// TwinCAT 3 PLC project PLC1
// Company: Nibe Airsite
// ProgramVersion: 3.1.4024.12
// libraries:
//   Tc2_DataExchange, * (Beckhoff Automation GmbH)
//   Tc2_ModbusRTU, * (Beckhoff Automation GmbH)
//   Tc2_ModbusSrv, * (Beckhoff Automation GmbH)
//   Tc2_Standard, * (Beckhoff Automation GmbH)
//   Tc2_SUPS, * (Beckhoff Automation GmbH)
//   Tc2_System, * (Beckhoff Automation GmbH)
//   Tc2_SystemCX, * (Beckhoff Automation GmbH)
//   Tc2_TcpIp, * (Beckhoff Automation GmbH)
//   Tc2_Utilities, * (Beckhoff Automation GmbH)
//   Tc3_BA_Common, * (Beckhoff Automation GmbH)
//   Tc3_JsonXml, * (Beckhoff Automation GmbH)
//   Tc3_Module, * (Beckhoff Automation GmbH)
// project tree:
//   DUTs/Alarms/ AlarmDef.TcDUT, AlarmHandler.TcPOU, AlarmPolarity.TcDUT, AlarmPriority.TcDUT, AlarmLog.TcDUT, AlarmMonitor.TcPOU, AlarmEvent.TcDUT
//   DUTs/Custom/ExtraAlarms/ AdsTagsExtraAlarms.TcDUT, GreenMasterStatusExtraAlarms.TcDUT, ExtraAlarms_Interface.TcPOU
//   DUTs/Custom/ParallelUnits/ AdsTagsParallelUnits.TcDUT, ParallelUnits.TcPOU, ParallelUnitsSettings.TcDUT, ParallelUnitsStatus.TcDUT, RemoteOrder.TcDUT, RemoteStatusData.TcDUT
//   DUTs/Custom/SmokeControl/ AdsTagsSmokeControl.TcDUT, SmokeControl_Interface.TcPOU, GreenMasterStatusSmokeControl.TcDUT, SxDuoInterface.TcDUT
//   DUTs/Custom/Redundancy/ TagsRedundancy.TcDUT (not stored), adsValue_AggStat.TcPOU, AggStat.TcDUT, RedundancyStatus.TcDUT, RedundancySettings.TcDUT (not stored), Redundancy.TcPOU
//   DUTs/Custom/_Standard/ AdsTags.TcDUT, GreenMasterSettings.TcDUT, GreenMasterStatus.TcDUT, Standard_Interface.TcPOU, TimeChannel_CT_CF.TcDUT
//   DUTs/Defrost/ DefrostSections.TcDUT, Defrost.TcPOU, DefrostStates.TcDUT
//   DUTs/Exercise/ ExerciseF_QM2.TcPOU, ExerciseF_P1.TcPOU
//   DUTs/GreenMaster/ SystemStatesRunMode.TcDUT, SystemStatesRunModeExternal.TcDUT, GreenMasterXXL.TcPOU, GreenMasterBase.TcPOU, SystemStates.TcDUT
//   DUTs/IO/ AI3468.TcDUT, AnalogInput.TcPOU, FlowInput.TcPOU, TemperatureInput.TcPOU, AnalogOutput.TcPOU, AnalogSwitch.TcPOU, DigitalInput.TcPOU, DigitalOutput.TcPOU, BaseIO.TcPOU, PressureInput.TcPOU, TIoKind.TcDUT
//   DUTs/ModbusRTU/ EBM_Speed.TcPOU, Gebhardt_Power.TcPOU, Gebhardt_Speed.TcPOU, ModbusReadWordArray.TcPOU, EBM_Power.TcPOU, Modbus.TcPOU, ModbusIo.TcPOU, ModbusWriteBits.TcPOU, ModbusWriteWord.TcPOU, ModbusRegisterType.TcDUT, ModbusRTU.TcPOU, ModbusReadWord.TcPOU, ModbusReadBits.TcPOU
//   DUTs/Parameters/Alarm/ AlarmControl.TcDUT, AlarmDelays.TcDUT, AlarmLimits.TcDUT, AlarmLimitsA.TcDUT, AlarmLimitsB.TcDUT, AlarmLimitsC.TcDUT, AlarmParameters.TcDUT, AlarmParametersFB.TcPOU (not stored), AlarmsA.TcDUT, AlarmsB.TcDUT, AlarmsC.TcDUT, AlarmsDelaysA.TcDUT, AlarmsDelaysB.TcDUT, AlarmsDelaysC.TcDUT, AlarmSignals.TcDUT
//   DUTs/Controllers/ Band.TcPOU, BandLimit.TcPOU, Controller.TcPOU, PidController.TcPOU, InterpolateNewton.TcPOU, Interpolate.TcPOU, Ramp.TcPOU
//   DUTs/Controls/ SupplyAirControl.TcPOU, ExtractAirControl.TcPOU
//   DUTs/Dampers/ BaseDamper.TcPOU, Damper.TcPOU, DamperMonitor.TcPOU
//   DUTs/Events/ Event.TcDUT, EventLog.TcPOU, EventLogData.TcDUT, EventTypes.TcDUT
//   DUTs/Fans/ Fan.TcPOU, FanControl.TcPOU, FanControlTypes.TcDUT, PostVentilation.TcPOU, PressureToFlow.TcPOU, SpecificFanPower.TcPOU
//   DUTs/Fire/ FireDamper.TcPOU, SmokeDetector.TcPOU
//   DUTs/GreenMaster/IO/ GreenMasterAIU_Base.TcPOU, GreenMasterAIU_ModbusRTU.TcPOU, GreenMasterAI_Base.TcPOU, GreenMasterAO_Base.TcPOU, GreenMasterDI_Base.TcPOU, GreenMasterDO_Base.TcPOU, GreenMasterSmokeControl.TcPOU, GreenMasterSmokeControl_Base.TcPOU, GreenMasterAI.TcPOU, GreenMasterAIU.TcPOU, GreenMasterAO.TcPOU, GreenMasterDI.TcPOU, GreenMasterDO.TcPOU
//   DUTs/ModbusTCP/ ModbusTCP.TcPOU
//   DUTs/Parameters/ GreenMasterBaseParameters.TcDUT, GreenMasterBaseParametersFB.TcPOU, GreenMasterParametersXXL.TcDUT, GreenMasterParametersXXLFB.TcDUT
//   DUTs/Parameters/IO/ AnalogInputParameters.TcDUT, AnalogInputParametersFB.TcPOU, AnalogOutputCalibration.TcDUT, AnalogOutputCalibrationParameters.TcDUT, AnalogOutputOverrideParameters.TcDUT, AnalogOutputParameters.TcDUT, AnalogOutputParametersFB.TcPOU, DigitalInputParameters.TcDUT, DigitalInputParametersFB.TcPOU, DigitalOutputOverrideParameters.TcDUT, DigitalOutputParameters.TcDUT, DigitalOutputParametersFB.TcPOU, InputStatus.TcDUT, IoParameters.TcDUT, IOParametersFB.TcPOU, IoStatus.TcDUT, SensorStatus.TcDUT, SmokeControlStatus.TcDUT
//   DUTs/Parameters/Redundancy/ RedundancyParameters.TcDUT
//   DUTs/Parameters/Regulation/ AirParameters.TcDUT, AirParametersFB.TcPOU, ColdRecyclingParameters.TcDUT, ControllerParameters.TcDUT, DefaultParameters.TcDUT, DefaultParametersFB.TcPOU, FanTypes.TcDUT, FireParameters.TcDUT, HeaterOutputDirections.TcDUT, RegulationControlParameters.TcDUT, RegulationParameters.TcDUT, RegulationParametersFB.TcPOU, SetPointAdjustment.TcDUT, SetPointAdjustmentFB.TcPOU, SetPointOffsetCurve.TcDUT, TemperatureCompensationSources.TcDUT, TemperatureControlParameters.TcDUT, TemperatureControlParametersFB.TcPOU, TemperatureControlSources.TcDUT
//   DUTs/Parameters/Simulation/ SimulateFlow.TcPOU, SimulationFB.TcPOU, SimulationParameters.TcDUT, SimulationParametersFB.TcPOU
//   DUTs/Parameters/SmokeControl/ NetLinkParameters.TcDUT, NetLinkParametersFB.TcPOU, SmokeControlExerciseParameters.TcDUT, SmokeControlFireParameters.TcDUT, SmokeControlParametersBase.TcDUT, SmokeControlParametersBaseFB.TcPOU, SxDuoCommand.TcDUT, SxDuoParameters.TcDUT, SxDuoParametersFB.TcPOU, SxDuoStatus.TcDUT, SxDuoUnit.TcDUT, SxDuoUnitFB.TcPOU
//   DUTs/Parameters/System/Defrost/ DefrostParameters.TcDUT, DefrostStageParameters.TcDUT, SetPointReductionParameters.TcDUT, WinterShutdownParameters.TcDUT
//   DUTs/Parameters/System/Exercise/ ExerciseCirculationPumpsParameters.TcDUT, ExerciseCirculationPumpsParametersFB.TcPOU, ExerciseExternalFireControlParameters.TcDUT, ExerciseExternalFireControlParametersFB.TcPOU, ExerciseFireBypassDamperParameters.TcDUT, ExerciseFireBypassDamperParametersFB.TcPOU, ExerciseParameters.TcDUT, ExerciseParametersFB.TcPOU
//   DUTs/Parameters/System/Operation/ AlternativeOperation.TcDUT, CoolingRecycling.TcDUT, DIStartUnit.TcDUT, LocalTimeControl.TcDUT, MaxFilterPressure.TcDUT, NightReduction.TcDUT, OperationParametersFB.TcPOU, OvkActivation.TcDUT, RecirculationControl.TcDUT, RelativeHumidity.TcDUT, SetPointTypes.TcDUT, StartControl.TcDUT, StartupFanDelay.TcDUT, StartupRecycling.TcDUT, SystemOperationParameters.TcDUT, SystemOperationParametersXXL.TcDUT, TimeChannelDayParameters.TcDUT, TimeChannelParameters.TcDUT, TimeChannelParametersFB.TcPOU, TimeChannelDayParametersFB.TcPOU, UnitOperation.TcDUT
//   DUTs/Parameters/System/ SystemParameters.TcDUT, SystemParametersFB.TcPOU, SystemParametersXXL.TcDUT
//   DUTs/Smoke Control/ DamperControl.TcPOU, DamperModule.TcPOU
//   DUTs/System/ AnyEqual.TcPOU, Permissions.TcDUT, Supervisor.TcPOU, User.TcDUT
//   DUTs/Utilities/ ActuatorMonitor.TcPOU, AnalogMultiplexer.TcPOU, Average.TcPOU, DeviationMonitor.TcPOU, DeviationMonitorMode.TcDUT, CalculateEfficiency.TcPOU, ifc_int.TcPOU, ifc_bool.TcPOU, ifc_lreal.TcPOU, LREAL_BMUX.TcPOU, BOOL_BMUX.TcPOU, BoolToErrorText.TcPOU, DigitalSignal.TcPOU, EMA.TcPOU, GetBit.TcPOU, GetTickCount.TcPOU, Hysteresis.TcPOU, LimitValue.TcPOU, MAX_FB.TcPOU, MIN_FB.TcPOU, NowDT.TcPOU, PulseCounter.TcPOU, PWM.TcPOU, REAL_TO_WORD_SAFE.TcPOU, LREAL_TO_WORD_SAFE.TcPOU, Scale.TcPOU, SetBit.TcPOU, TimeChannel1CH.TcPOU, TimeChannel1CH_Data.TcDUT, TimeChannelSettings.TcDUT, Timer.TcPOU, TimerDays.TcDUT, WriteBoolIf.TcPOU, WriteLRealIf.TcPOU, WriteLRealOnlyIf.TcPOU
//   DUTs/Valves/ BaseValve.TcPOU, Valve.TcPOU, ValveMonitor.TcPOU
//   DUTs/Ventilation/ FB_GM_NIGHTCOOL.TcPOU, VentilationControl.TcPOU
//   GVLs/ ADS_ParallelUnits.TcGVL, ADS_SmokeControl.TcGVL, ADS_Standard.TcGVL, ADS_ExtraAlarms.TcGVL, AnalogInputs.TcDUT, AnalogOutputs.TcDUT, DigitalInputs.TcDUT, DigitalInputLevels.TcDUT, DigitalOutputs.TcDUT, ComponentNames.TcDUT, ExtraAlarmInputs.TcGVL, GetComponent.TcPOU, Globals.TcGVL, GVL.TcGVL, GVL_Redundancy.TcGVL, IOTypes.TcDUT, GlobalSettings.TcGVL, Component.TcDUT, ModbusRTU_IO.TcDUT
//   / PlcTask.TcTTO, Task_4.TcTTO
//   POUs/ AdsWriteVariable.TcPOU, GreenMasterXXL_FB.TcPOU, Main.TcPOU, SimpleTimeChannel.TcPOU, SmokeControl.TcPOU, AdsReadVariable.TcPOU, TestPID.TcPOU, Timers.TcPOU
// real-time tasks:
//   TASK PlcTask: cycle T#50000us, priority 20, ADS port 350
//   TASK Task 4: cycle T#10ms, priority 1, ADS port 351
// I/O:
//   DEVICE Device 1 (Beckhoff CCAT)
//   DEVICE Device CTH (CX-BK) (disabled)
//     Box CTH (CX-BK)
//   DEVICE Device STD (CX-BK)
//     Box STD (CX-BK)
//   DEVICE Device GMA (CX-BK) (disabled)
//     Box STD (CX-BK)
// variable links:
//   PLC1/PLC1 Instance <-> Device CTH (CX-BK)/Box CTH (CX-BK)
//     PlcTask Inputs/Globals.IO.AIn.AI01_Error <-> AI 2.1 (KL3208-0010-4)/Channel 1/State @bit 6
//     PlcTask Inputs/Globals.IO.AIn.AI02_Error <-> AI 2.1 (KL3208-0010-4)/Channel 2/State @bit 6
//     PlcTask Inputs/Globals.IO.AIn.AI03_Error <-> AI 2.1 (KL3208-0010-4)/Channel 3/State @bit 6
//     PlcTask Inputs/Globals.IO.AIn.AI04_Error <-> AI 2.1 (KL3208-0010-4)/Channel 4/State @bit 6
//     PlcTask Inputs/Globals.IO.AIn.AI05_Error <-> AI 2.2 (KL3208-0010-4)/Channel 1/State @bit 6
//     PlcTask Inputs/Globals.IO.AIn.AI06_Error <-> AI 2.2 (KL3208-0010-4)/Channel 2/State @bit 6
//     PlcTask Inputs/Globals.IO.AIn.AI07_Error <-> AI 2.2 (KL3208-0010-4)/Channel 3/State @bit 6
//     PlcTask Inputs/Globals.IO.AIn.AI08_Error <-> AI 2.2 (KL3208-0010-4)/Channel 4/State @bit 6
//     PlcTask Inputs/Globals.IO.AIn.AI09_Error <-> AI 3.1 (KL3208-0010-4)/Channel 1/State @bit 6
//     PlcTask Inputs/Globals.IO.AIn.AI10_Error <-> AI 3.1 (KL3208-0010-4)/Channel 2/State @bit 6
//     PlcTask Inputs/Globals.IO.AIn.AI11_Error <-> AI 3.1 (KL3208-0010-4)/Channel 3/State @bit 6
//     PlcTask Inputs/Globals.IO.AIn.AI12_Error <-> AI 3.1 (KL3208-0010-4)/Channel 4/State @bit 6
//     PlcTask Inputs/Globals.IO.AIn.AI13_Error <-> AI 3.2 (KL3208-0010-4)/Channel 1/State @bit 6
//     PlcTask Inputs/Globals.IO.AIn.AI14_Error <-> AI 3.2 (KL3208-0010-4)/Channel 2/State @bit 6
//     PlcTask Inputs/Globals.IO.AIn.AI15_Error <-> AI 3.2 (KL3208-0010-4)/Channel 3/State @bit 6
//     PlcTask Inputs/Globals.IO.AIn.AI16_Error <-> AI 3.2 (KL3208-0010-4)/Channel 4/State @bit 6
//     PlcTask Inputs/Globals.IO.AIn.AI17_Error <-> AI 4.1 (KL3468-4)/Channel 1/State @bit 6
//     PlcTask Inputs/Globals.IO.AIn.AI18_Error <-> AI 4.1 (KL3468-4)/Channel 2/State @bit 6
//     PlcTask Inputs/Globals.IO.AIn.AI19_Error <-> AI 4.1 (KL3468-4)/Channel 3/State @bit 6
//     PlcTask Inputs/Globals.IO.AIn.AI20_Error <-> AI 4.1 (KL3468-4)/Channel 4/State @bit 6
//     PlcTask Inputs/Globals.IO.AIn.AI21_Error <-> AI 4.2 (KL3468-4)/Channel 1/State @bit 6
//     PlcTask Inputs/Globals.IO.AIn.AI22_Error <-> AI 4.2 (KL3468-4)/Channel 2/State @bit 6
//     PlcTask Inputs/Globals.IO.AIn.AI23_Error <-> AI 4.2 (KL3468-4)/Channel 3/State @bit 6
//     PlcTask Inputs/Globals.IO.AIn.AI24_Error <-> AI 4.2 (KL3468-4)/Channel 4/State @bit 6
//     PlcTask Inputs/Globals.IO.DIn.DI01 <-> DI 1 (KL1408)/Channel 1/Input
//     PlcTask Inputs/Globals.IO.DIn.DI02 <-> DI 1 (KL1408)/Channel 2/Input
//     PlcTask Inputs/Globals.IO.DIn.DI03 <-> DI 1 (KL1408)/Channel 3/Input
//     PlcTask Inputs/Globals.IO.DIn.DI04 <-> DI 1 (KL1408)/Channel 4/Input
//     PlcTask Inputs/Globals.IO.DIn.DI05 <-> DI 1 (KL1408)/Channel 5/Input
//     PlcTask Inputs/Globals.IO.DIn.DI06 <-> DI 1 (KL1408)/Channel 6/Input
//     PlcTask Inputs/Globals.IO.DIn.DI07 <-> DI 1 (KL1408)/Channel 7/Input
//     PlcTask Inputs/Globals.IO.DIn.DI08 <-> DI 1 (KL1408)/Channel 8/Input
//     PlcTask Inputs/Globals.IO.DIn.DI09 <-> DI 2 (KL1408)/Channel 1/Input
//     PlcTask Inputs/Globals.IO.DIn.DI10 <-> DI 2 (KL1408)/Channel 2/Input
//     PlcTask Inputs/Globals.IO.DIn.DI11 <-> DI 2 (KL1408)/Channel 3/Input
//     PlcTask Inputs/Globals.IO.DIn.DI12 <-> DI 2 (KL1408)/Channel 4/Input
//     PlcTask Inputs/Globals.IO.DIn.DI13 <-> DI 2 (KL1408)/Channel 5/Input
//     PlcTask Inputs/Globals.IO.DIn.DI14 <-> DI 2 (KL1408)/Channel 6/Input
//     PlcTask Inputs/Globals.IO.DIn.DI15 <-> DI 2 (KL1408)/Channel 7/Input
//     PlcTask Inputs/Globals.IO.DIn.DI16 <-> DI 2 (KL1408)/Channel 8/Input
//     PlcTask Inputs/Globals.IO.DIn.DI17 <-> DI 3 (KL1408)/Channel 1/Input
//     PlcTask Inputs/Globals.IO.DIn.DI18 <-> DI 3 (KL1408)/Channel 2/Input
//     PlcTask Inputs/Globals.IO.DIn.DI19 <-> DI 3 (KL1408)/Channel 3/Input
//     PlcTask Inputs/Globals.IO.DIn.DI20 <-> DI 3 (KL1408)/Channel 4/Input
//     PlcTask Inputs/Globals.IO.DIn.DI21 <-> DI 3 (KL1408)/Channel 5/Input
//     PlcTask Inputs/Globals.IO.DIn.DI22 <-> DI 3 (KL1408)/Channel 6/Input
//     PlcTask Inputs/Globals.IO.DIn.DI23 <-> DI 3 (KL1408)/Channel 7/Input
//     PlcTask Inputs/Globals.IO.DIn.DI24 <-> DI 3 (KL1408)/Channel 8/Input
//     PlcTask Outputs/Globals.IO.AOut.AO01 <-> AO 1.1 (KL4408-4)/Channel 1/Data Out
//     PlcTask Outputs/Globals.IO.AOut.AO02 <-> AO 1.1 (KL4408-4)/Channel 2/Data Out
//     PlcTask Outputs/Globals.IO.AOut.AO03 <-> AO 1.1 (KL4408-4)/Channel 3/Data Out
//     PlcTask Outputs/Globals.IO.AOut.AO04 <-> AO 1.1 (KL4408-4)/Channel 4/Data Out
//     PlcTask Outputs/Globals.IO.AOut.AO05 <-> AO 1.2 (KL4408-4)/Channel 1/Data Out
//     PlcTask Outputs/Globals.IO.AOut.AO06 <-> AO 1.2 (KL4408-4)/Channel 2/Data Out
//     PlcTask Outputs/Globals.IO.AOut.AO07 <-> AO 1.2 (KL4408-4)/Channel 3/Data Out
//     PlcTask Outputs/Globals.IO.AOut.AO08 <-> AO 1.2 (KL4408-4)/Channel 4/Data Out
//     PlcTask Outputs/Globals.IO.DOut.DO01 <-> DO 1 (KL2408)/Channel 1/Output
//     PlcTask Outputs/Globals.IO.DOut.DO02 <-> DO 1 (KL2408)/Channel 2/Output
//     PlcTask Outputs/Globals.IO.DOut.DO03 <-> DO 1 (KL2408)/Channel 3/Output
//     PlcTask Outputs/Globals.IO.DOut.DO04 <-> DO 1 (KL2408)/Channel 4/Output
//     PlcTask Outputs/Globals.IO.DOut.DO05 <-> DO 1 (KL2408)/Channel 5/Output
//     PlcTask Outputs/Globals.IO.DOut.DO06 <-> DO 1 (KL2408)/Channel 6/Output
//     PlcTask Outputs/Globals.IO.DOut.DO07 <-> DO 1 (KL2408)/Channel 7/Output
//     PlcTask Outputs/Globals.IO.DOut.DO08 <-> DO 1 (KL2408)/Channel 8/Output
//     PlcTask Outputs/Globals.IO.DOut.DO09 <-> DO 2 (KL2408)/Channel 1/Output
//     PlcTask Outputs/Globals.IO.DOut.DO10 <-> DO 2 (KL2408)/Channel 2/Output
//     PlcTask Outputs/Globals.IO.DOut.DO11 <-> DO 2 (KL2408)/Channel 3/Output
//     PlcTask Outputs/Globals.IO.DOut.DO12 <-> DO 2 (KL2408)/Channel 4/Output
//     PlcTask Outputs/Globals.IO.DOut.DO13 <-> DO 2 (KL2408)/Channel 5/Output
//     PlcTask Outputs/Globals.IO.DOut.DO14 <-> DO 2 (KL2408)/Channel 6/Output
//     PlcTask Outputs/Globals.IO.DOut.DO15 <-> DO 2 (KL2408)/Channel 7/Output
//     PlcTask Outputs/Globals.IO.DOut.DO16 <-> DO 2 (KL2408)/Channel 8/Output
//     PlcTask Outputs/Globals.IO.DOut.RDO01 <-> RDO 1 (KL2652)/Channel 1/Output
//     PlcTask Outputs/Globals.IO.DOut.RDO02 <-> RDO 1 (KL2652)/Channel 2/Output
//     PlcTask Outputs/Globals.IO.DOut.RDO03 <-> RDO 2 (KL2652)/Channel 1/Output
//     PlcTask Outputs/Globals.IO.DOut.RDO04 <-> RDO 2 (KL2652)/Channel 2/Output
//   PLC1/PLC1 Instance <-> Device GMA (CX-BK)/Box STD (CX-BK)
//     PlcTask Inputs/Globals.IO.AIn.AI01_Error <-> AI 2.1 (KL3208-0010-4)/Channel 1/State @bit 6
//     PlcTask Inputs/Globals.IO.AIn.AI02_Error <-> AI 2.1 (KL3208-0010-4)/Channel 2/State @bit 6
//     PlcTask Inputs/Globals.IO.AIn.AI03_Error <-> AI 2.1 (KL3208-0010-4)/Channel 3/State @bit 6
//     PlcTask Inputs/Globals.IO.AIn.AI04_Error <-> AI 2.1 (KL3208-0010-4)/Channel 4/State @bit 6
//     PlcTask Inputs/Globals.IO.AIn.AI05_Error <-> AI 2.2 (KL3208-0010-4)/Channel 1/State @bit 6
//     PlcTask Inputs/Globals.IO.AIn.AI06_Error <-> AI 2.2 (KL3208-0010-4)/Channel 2/State @bit 6
//     PlcTask Inputs/Globals.IO.AIn.AI07_Error <-> AI 2.2 (KL3208-0010-4)/Channel 3/State @bit 6
//     PlcTask Inputs/Globals.IO.AIn.AI08_Error <-> AI 2.2 (KL3208-0010-4)/Channel 4/State @bit 6
//     PlcTask Inputs/Globals.IO.DIn.DI01 <-> DI 1 (KL1408)/Channel 1/Input
//     PlcTask Inputs/Globals.IO.DIn.DI02 <-> DI 1 (KL1408)/Channel 2/Input
//     PlcTask Inputs/Globals.IO.DIn.DI03 <-> DI 1 (KL1408)/Channel 3/Input
//     PlcTask Inputs/Globals.IO.DIn.DI04 <-> DI 1 (KL1408)/Channel 4/Input
//     PlcTask Inputs/Globals.IO.DIn.DI05 <-> DI 1 (KL1408)/Channel 5/Input
//     PlcTask Inputs/Globals.IO.DIn.DI06 <-> DI 1 (KL1408)/Channel 6/Input
//     PlcTask Inputs/Globals.IO.DIn.DI07 <-> DI 1 (KL1408)/Channel 7/Input
//     PlcTask Inputs/Globals.IO.DIn.DI08 <-> DI 1 (KL1408)/Channel 8/Input
//     PlcTask Inputs/Globals.IO.DIn.DI09 <-> DI 2 (KL1408)/Channel 1/Input
//     PlcTask Inputs/Globals.IO.DIn.DI10 <-> DI 2 (KL1408)/Channel 2/Input
//     PlcTask Inputs/Globals.IO.DIn.DI11 <-> DI 2 (KL1408)/Channel 3/Input
//     PlcTask Inputs/Globals.IO.DIn.DI12 <-> DI 2 (KL1408)/Channel 4/Input
//     PlcTask Inputs/Globals.IO.DIn.DI13 <-> DI 2 (KL1408)/Channel 5/Input
//     PlcTask Inputs/Globals.IO.DIn.DI14 <-> DI 2 (KL1408)/Channel 6/Input
//     PlcTask Inputs/Globals.IO.DIn.DI15 <-> DI 2 (KL1408)/Channel 7/Input
//     PlcTask Inputs/Globals.IO.DIn.DI16 <-> DI 2 (KL1408)/Channel 8/Input
//     PlcTask Outputs/Globals.IO.AOut.AO01 <-> AO 1.1 (KL4408-4)/Channel 1/Data Out
//     PlcTask Outputs/Globals.IO.AOut.AO02 <-> AO 1.1 (KL4408-4)/Channel 2/Data Out
//     PlcTask Outputs/Globals.IO.AOut.AO03 <-> AO 1.1 (KL4408-4)/Channel 3/Data Out
//     PlcTask Outputs/Globals.IO.AOut.AO04 <-> AO 1.1 (KL4408-4)/Channel 4/Data Out
//     PlcTask Outputs/Globals.IO.AOut.AO05 <-> AO 1.2 (KL4408-4)/Channel 1/Data Out
//     PlcTask Outputs/Globals.IO.AOut.AO06 <-> AO 1.2 (KL4408-4)/Channel 2/Data Out
//     PlcTask Outputs/Globals.IO.AOut.AO07 <-> AO 1.2 (KL4408-4)/Channel 3/Data Out
//     PlcTask Outputs/Globals.IO.AOut.AO08 <-> AO 1.2 (KL4408-4)/Channel 4/Data Out
//     PlcTask Outputs/Globals.IO.DOut.DO01 <-> DO 1 (KL2408)/Channel 1/Output
//     PlcTask Outputs/Globals.IO.DOut.DO02 <-> DO 1 (KL2408)/Channel 2/Output
//     PlcTask Outputs/Globals.IO.DOut.DO03 <-> DO 1 (KL2408)/Channel 3/Output
//     PlcTask Outputs/Globals.IO.DOut.DO04 <-> DO 1 (KL2408)/Channel 4/Output
//     PlcTask Outputs/Globals.IO.DOut.DO05 <-> DO 1 (KL2408)/Channel 5/Output
//     PlcTask Outputs/Globals.IO.DOut.DO06 <-> DO 1 (KL2408)/Channel 6/Output
//     PlcTask Outputs/Globals.IO.DOut.DO07 <-> DO 1 (KL2408)/Channel 7/Output
//     PlcTask Outputs/Globals.IO.DOut.DO08 <-> DO 1 (KL2408)/Channel 8/Output
//     PlcTask Outputs/Globals.IO.DOut.RDO01 <-> RDO 1 (KL2652)/Channel 1/Output
//     PlcTask Outputs/Globals.IO.DOut.RDO02 <-> RDO 1 (KL2652)/Channel 2/Output
//     PlcTask Outputs/Globals.IO.DOut.RDO03 <-> RDO 2 (KL2652)/Channel 1/Output
//     PlcTask Outputs/Globals.IO.DOut.RDO04 <-> RDO 2 (KL2652)/Channel 2/Output
//   PLC1/PLC1 Instance <-> Device STD (CX-BK)/Box STD (CX-BK)
//     PlcTask Inputs/ExtraAlarmInputs.AL01 <-> DI 3 (KL1408)/Channel 1/Input
//     PlcTask Inputs/ExtraAlarmInputs.AL02 <-> DI 3 (KL1408)/Channel 2/Input
//     PlcTask Inputs/ExtraAlarmInputs.AL03 <-> DI 3 (KL1408)/Channel 3/Input
//     PlcTask Inputs/ExtraAlarmInputs.AL04 <-> DI 3 (KL1408)/Channel 4/Input
//     PlcTask Inputs/ExtraAlarmInputs.AL05 <-> DI 3 (KL1408)/Channel 5/Input
//     PlcTask Inputs/ExtraAlarmInputs.AL06 <-> DI 3 (KL1408)/Channel 6/Input
//     PlcTask Inputs/ExtraAlarmInputs.AL07 <-> DI 3 (KL1408)/Channel 7/Input
//     PlcTask Inputs/ExtraAlarmInputs.AL08 <-> DI 3 (KL1408)/Channel 8/Input
//     PlcTask Inputs/Globals.AI3468.AI1 <-> AI 2.3 (KL3468-4)/Channel 1/Data In
//     PlcTask Inputs/Globals.AI3468.AI2 <-> AI 2.3 (KL3468-4)/Channel 2/Data In
//     PlcTask Inputs/Globals.IO.AIn.AI01 <-> AI 2.1 (KL3208-0010-4)/Channel 1/Data In
//     PlcTask Inputs/Globals.IO.AIn.AI02 <-> AI 2.1 (KL3208-0010-4)/Channel 2/Data In
//     PlcTask Inputs/Globals.IO.AIn.AI03 <-> AI 2.1 (KL3208-0010-4)/Channel 3/Data In
//     PlcTask Inputs/Globals.IO.AIn.AI04 <-> AI 2.1 (KL3208-0010-4)/Channel 4/Data In
//     PlcTask Inputs/Globals.IO.AIn.AI05 <-> AI 2.2 (KL3208-0010-4)/Channel 1/Data In
//     PlcTask Inputs/Globals.IO.AIn.AI06 <-> AI 2.2 (KL3208-0010-4)/Channel 2/Data In
//     PlcTask Inputs/Globals.IO.AIn.AI07 <-> AI 2.2 (KL3208-0010-4)/Channel 3/Data In
//     PlcTask Inputs/Globals.IO.AIn.AI08 <-> AI 2.2 (KL3208-0010-4)/Channel 4/Data In
//     PlcTask Inputs/Globals.IO.AIn.AI01_Error <-> AI 2.1 (KL3208-0010-4)/Channel 1/State @bit 6
//     PlcTask Inputs/Globals.IO.AIn.AI02_Error <-> AI 2.1 (KL3208-0010-4)/Channel 2/State @bit 6
//     PlcTask Inputs/Globals.IO.AIn.AI03_Error <-> AI 2.1 (KL3208-0010-4)/Channel 3/State @bit 6
//     PlcTask Inputs/Globals.IO.AIn.AI04_Error <-> AI 2.1 (KL3208-0010-4)/Channel 4/State @bit 6
//     PlcTask Inputs/Globals.IO.AIn.AI05_Error <-> AI 2.2 (KL3208-0010-4)/Channel 1/State @bit 6
//     PlcTask Inputs/Globals.IO.AIn.AI06_Error <-> AI 2.2 (KL3208-0010-4)/Channel 2/State @bit 6
//     PlcTask Inputs/Globals.IO.AIn.AI07_Error <-> AI 2.2 (KL3208-0010-4)/Channel 3/State @bit 6
//     PlcTask Inputs/Globals.IO.AIn.AI08_Error <-> AI 2.2 (KL3208-0010-4)/Channel 4/State @bit 6
//     PlcTask Inputs/Globals.IO.AIn.AI09 <-> Inputs/State
//     PlcTask Inputs/Globals.IO.DIn.DI01 <-> DI 1 (KL1408)/Channel 1/Input
//     PlcTask Inputs/Globals.IO.DIn.DI02 <-> DI 1 (KL1408)/Channel 2/Input
//     PlcTask Inputs/Globals.IO.DIn.DI03 <-> DI 1 (KL1408)/Channel 3/Input
//     PlcTask Inputs/Globals.IO.DIn.DI04 <-> DI 1 (KL1408)/Channel 4/Input
//     PlcTask Inputs/Globals.IO.DIn.DI05 <-> DI 1 (KL1408)/Channel 5/Input
//     PlcTask Inputs/Globals.IO.DIn.DI06 <-> DI 1 (KL1408)/Channel 6/Input
//     PlcTask Inputs/Globals.IO.DIn.DI07 <-> DI 1 (KL1408)/Channel 7/Input
//     PlcTask Inputs/Globals.IO.DIn.DI08 <-> DI 1 (KL1408)/Channel 8/Input
//     PlcTask Inputs/Globals.IO.DIn.DI09 <-> DI 2 (KL1408)/Channel 1/Input
//     PlcTask Inputs/Globals.IO.DIn.DI10 <-> DI 2 (KL1408)/Channel 2/Input
//     PlcTask Inputs/Globals.IO.DIn.DI11 <-> DI 2 (KL1408)/Channel 3/Input
//     PlcTask Inputs/Globals.IO.DIn.DI12 <-> DI 2 (KL1408)/Channel 4/Input
//     PlcTask Inputs/Globals.IO.DIn.DI13 <-> DI 2 (KL1408)/Channel 5/Input
//     PlcTask Inputs/Globals.IO.DIn.DI14 <-> DI 2 (KL1408)/Channel 6/Input
//     PlcTask Inputs/Globals.IO.DIn.DI15 <-> DI 2 (KL1408)/Channel 7/Input
//     PlcTask Inputs/Globals.IO.DIn.DI16 <-> DI 2 (KL1408)/Channel 8/Input
//     PlcTask Inputs/Main.GreenMasterAI2_RTU.ModbusRTU.ModbusMaster.InData/D <-> Modbus RTU (KL6041)/Channel 1/Data In 0
//     PlcTask Inputs/Main.GreenMasterAI2_RTU.ModbusRTU.ModbusMaster.InData/D @bit {8..168 step 8} <-> Modbus RTU (KL6041)/Channel 1/Data In {1..21}  (21 links)
//     PlcTask Inputs/Main.GreenMasterAI2_RTU.ModbusRTU.ModbusMaster.InData/Status <-> Modbus RTU (KL6041)/Channel 1/State
//     PlcTask Outputs/Globals.IO.AOut.AO01 <-> AO 1.1 (KL4408-4)/Channel 1/Data Out
//     PlcTask Outputs/Globals.IO.AOut.AO02 <-> AO 1.1 (KL4408-4)/Channel 2/Data Out
//     PlcTask Outputs/Globals.IO.AOut.AO03 <-> AO 1.1 (KL4408-4)/Channel 3/Data Out
//     PlcTask Outputs/Globals.IO.AOut.AO04 <-> AO 1.1 (KL4408-4)/Channel 4/Data Out
//     PlcTask Outputs/Globals.IO.AOut.AO05 <-> AO 1.2 (KL4408-4)/Channel 1/Data Out
//     PlcTask Outputs/Globals.IO.AOut.AO06 <-> AO 1.2 (KL4408-4)/Channel 2/Data Out
//     PlcTask Outputs/Globals.IO.AOut.AO07 <-> AO 1.2 (KL4408-4)/Channel 3/Data Out
//     PlcTask Outputs/Globals.IO.AOut.AO08 <-> AO 1.2 (KL4408-4)/Channel 4/Data Out
//     PlcTask Outputs/Globals.IO.DOut.DO01 <-> DO 1 (KL2408)/Channel 1/Output
//     PlcTask Outputs/Globals.IO.DOut.DO02 <-> DO 1 (KL2408)/Channel 2/Output
//     PlcTask Outputs/Globals.IO.DOut.DO03 <-> DO 1 (KL2408)/Channel 3/Output
//     PlcTask Outputs/Globals.IO.DOut.DO04 <-> DO 1 (KL2408)/Channel 4/Output
//     PlcTask Outputs/Globals.IO.DOut.DO05 <-> DO 1 (KL2408)/Channel 5/Output
//     PlcTask Outputs/Globals.IO.DOut.DO06 <-> DO 1 (KL2408)/Channel 6/Output
//     PlcTask Outputs/Globals.IO.DOut.DO07 <-> DO 1 (KL2408)/Channel 7/Output
//     PlcTask Outputs/Globals.IO.DOut.DO08 <-> DO 1 (KL2408)/Channel 8/Output
//     PlcTask Outputs/Globals.IO.DOut.DO09 <-> DO 2 (KL2408)/Channel 1/Output
//     PlcTask Outputs/Globals.IO.DOut.DO10 <-> DO 2 (KL2408)/Channel 2/Output
//     PlcTask Outputs/Globals.IO.DOut.DO11 <-> DO 2 (KL2408)/Channel 3/Output
//     PlcTask Outputs/Globals.IO.DOut.DO12 <-> DO 2 (KL2408)/Channel 4/Output
//     PlcTask Outputs/Globals.IO.DOut.DO13 <-> DO 2 (KL2408)/Channel 5/Output
//     PlcTask Outputs/Globals.IO.DOut.DO14 <-> DO 2 (KL2408)/Channel 6/Output
//     PlcTask Outputs/Globals.IO.DOut.DO15 <-> DO 2 (KL2408)/Channel 7/Output
//     PlcTask Outputs/Globals.IO.DOut.DO16 <-> DO 2 (KL2408)/Channel 8/Output
//     PlcTask Outputs/Globals.IO.DOut.RDO01 <-> RDO 1 (KL2652)/Channel 1/Output
//     PlcTask Outputs/Globals.IO.DOut.RDO02 <-> RDO 1 (KL2652)/Channel 2/Output
//     PlcTask Outputs/Globals.IO.DOut.RDO03 <-> RDO 2 (KL2652)/Channel 1/Output
//     PlcTask Outputs/Globals.IO.DOut.RDO04 <-> RDO 2 (KL2652)/Channel 2/Output
//     PlcTask Outputs/Main.GreenMasterAI2_RTU.ModbusRTU.ModbusMaster.OutData/Ctrl <-> Modbus RTU (KL6041)/Channel 1/Ctrl
//     PlcTask Outputs/Main.GreenMasterAI2_RTU.ModbusRTU.ModbusMaster.OutData/D <-> Modbus RTU (KL6041)/Channel 1/Data Out 0
//     PlcTask Outputs/Main.GreenMasterAI2_RTU.ModbusRTU.ModbusMaster.OutData/D @bit {8..168 step 8} <-> Modbus RTU (KL6041)/Channel 1/Data Out {1..21}  (21 links)

CONFIGURATION PLC1
    RESOURCE PLC ON TwinCAT3
        TASK PlcTask(INTERVAL := T#50000us, PRIORITY := 20);
        TASK Task_4(INTERVAL := T#10ms, PRIORITY := 1);
        PROGRAM Main WITH PlcTask : Main;
        PROGRAM Timers WITH PlcTask : Timers;
    END_RESOURCE
END_CONFIGURATION

// ---- DUTs/Alarms/AlarmDef.TcDUT
TYPE AlarmDef :
STRUCT
	{attribute 'TcEncoding':='UTF-8'}
	Name: STRING;
	{attribute 'TcEncoding':='UTF-8'}
	Description: STRING;
	Active: BOOL;
	AutoReset: BOOL := TRUE;
	Delay: TIME := T#5S;
	EN: BOOL := TRUE;
	Value: LREAL;
	LimitValue: LREAL := 100;
	Polarity: AlarmPolarity := AlarmPolarity.ActiveHigh;
	Status: BOOL;
	Priority: AlarmPriority := AlarmPriority.A;
END_STRUCT
END_TYPE

// ---- DUTs/Alarms/AlarmPolarity.TcDUT
{attribute 'qualified_only'}
{attribute 'strict'}
TYPE AlarmPolarity :
(
	ActiveHigh := 0, ActiveLow
);
END_TYPE

// ---- DUTs/Alarms/AlarmPriority.TcDUT
{attribute 'qualified_only'}
{attribute 'strict'}
TYPE AlarmPriority :
(
	A := 0, B, C
);
END_TYPE

// ---- DUTs/Custom/ExtraAlarms/AdsTagsExtraAlarms.TcDUT
TYPE AdsTagsExtraAlarms :
STRUCT
	Status: GreenMasterStatusExtraAlarms;
END_STRUCT
END_TYPE

// ---- DUTs/Custom/ExtraAlarms/GreenMasterStatusExtraAlarms.TcDUT
TYPE GreenMasterStatusExtraAlarms :
STRUCT
	EXTRA_01_AL: BOOL; // Extra alarm 1
	EXTRA_02_AL: BOOL; // Extra alarm 2
	EXTRA_03_AL: BOOL; // Extra alarm 3
	EXTRA_04_AL: BOOL; // Extra alarm 4
	EXTRA_05_AL: BOOL; // Extra alarm 5
	EXTRA_06_AL: BOOL; // Extra alarm 6
	EXTRA_07_AL: BOOL; // Extra alarm 7
	EXTRA_08_AL: BOOL; // Extra alarm 8
END_STRUCT
END_TYPE

// ---- DUTs/Custom/ParallelUnits/AdsTagsParallelUnits.TcDUT
TYPE AdsTagsParallelUnits :
STRUCT
	Settings: ParallelUnitsSettings;
	Status: ParallelUnitsStatus;
END_STRUCT
END_TYPE

// ---- DUTs/Custom/ParallelUnits/ParallelUnitsSettings.TcDUT
TYPE ParallelUnitsSettings :
STRUCT
	RemoteAmsId: STRING := '5.73.47.143.1.1';
	PressureSupplySP: REAL := 0; // Set Point for Master/Slave
	PressureExtractSP: REAL := 0; // Set Point for Master/Slave
	PressureSupplySP_HighSpeed: REAL := 0; // Set Point for Master/Slave
	PressureExtractSP_HighSpeed: REAL := 0; // Set Point for Master/Slave
	SupplyAirSetPointAdjustment: SetPointAdjustment := (
		Curve := (Y1 := 250, Y2 := 250, Y3 := 250, Y4 := 250, Y5 := 250, Y6 := 250, Y7 := 250, Y8 := 250, Y9 := 250) 
	);
	ExtractAirSetPointAdjustment: SetPointAdjustment := (
		Curve := (Y1 := 250, Y2 := 250, Y3 := 250, Y4 := 250, Y5 := 250, Y6 := 250, Y7 := 250, Y8 := 250, Y9 := 250) 
	);
	StandaloneMaxFan: REAL := 0.7; // Max fan speed for single unit
	DualMinFan: REAL := 0.4; // Min fan speed for dual units
	Kp: REAL := 1.5; // P
	fTn: TIME := T#4M; // I time
	fTv: TIME := T#0M; // D time
	RemoteOrder: RemoteOrder;
END_STRUCT
END_TYPE

// ---- DUTs/Custom/ParallelUnits/ParallelUnitsStatus.TcDUT
TYPE ParallelUnitsStatus :
STRUCT
	PressureSupplyCSP: REAL; // Calculated Set Point for Master/Slave
	PressureExtractCSP: REAL; // Calculated Set Point for Master/Slave
	MasterActive: BOOL;
	IsMaster: BOOL;
	IsSlave: BOOL;
	SupplyFanSpeed: LREAL;
	ExtractFanSpeed: LREAL;
	IsRunning: BOOL;
	ResetAlarmMaster: BOOL;
	FireSupplyMaster: BOOL;
	FireExtractMaster: BOOL;
	FreezeMaster: BOOL;
	ResetAlarmSlave: BOOL;
	FireSupplySlave: BOOL;
	FireExtractSlave: BOOL;
	FreezeSlave: BOOL;
	State: SystemStates;
	CanBeRunnable: bool;
END_STRUCT
END_TYPE

// ---- DUTs/Custom/ParallelUnits/RemoteOrder.TcDUT
TYPE RemoteOrder :
STRUCT
	SupplySP: LREAL;
	ExtractSP: LREAL;
	DualSupplySP: LREAL;
	DualExtractSP: LREAL;
	DualSupplySP_HighSpeed: LREAL;
	DualExtractSP_HighSpeed: LREAL;
	Counter: INT;
	TimeChannels: TimeChannelParameters;
	TemperatureControl: ControllerParameters;
	TemperatureSetPointAdjustment: SetPointAdjustment; 
	SupplyAirSetPointAdjustment: SetPointAdjustment; 
	ExtractAirSetPointAdjustment: SetPointAdjustment; 
	NightCoolingRequest: BOOL;
END_STRUCT
END_TYPE

// ---- DUTs/Custom/ParallelUnits/RemoteStatusData.TcDUT
TYPE RemoteStatusData :
STRUCT
	Valid: BOOL;
	RemoteStatus: ParallelUnitsStatus;
END_STRUCT
END_TYPE

// ---- DUTs/Custom/SmokeControl/AdsTagsSmokeControl.TcDUT
TYPE AdsTagsSmokeControl :
STRUCT
	Status: GreenMasterStatusSmokeControl;
END_STRUCT
END_TYPE

// ---- DUTs/Custom/SmokeControl/GreenMasterStatusSmokeControl.TcDUT
TYPE GreenMasterStatusSmokeControl :
STRUCT
	COMM_AL: BOOL; // Communication alarm
	UNIT_01: SxDuoInterface;
	UNIT_02: SxDuoInterface;
	UNIT_03: SxDuoInterface;
	UNIT_04: SxDuoInterface;
	UNIT_05: SxDuoInterface;
	UNIT_06: SxDuoInterface;
	UNIT_07: SxDuoInterface;
	UNIT_08: SxDuoInterface;
	UNIT_09: SxDuoInterface;
	UNIT_10: SxDuoInterface;
	UNIT_11: SxDuoInterface;
	UNIT_12: SxDuoInterface;
	UNIT_13: SxDuoInterface;
	UNIT_14: SxDuoInterface;
	UNIT_15: SxDuoInterface;
END_STRUCT
END_TYPE

// ---- DUTs/Custom/Redundancy/AggStat.TcDUT
TYPE AggStat :
STRUCT
	SO1:BOOL;		// Serviceomkopplarläge 1 = service
	Driftfel:BOOL;	// Aggregatet är i driftfel eller
	TF_OP:REAL;		// Utsignal tilluftsfläkt
	TF_CMD:BOOL;	// Manöver tilluftsflöäkt
	FF_OP:REAL;		// Utsignal frånluftsfläkt
	FF_CMD:BOOL;	// Manöver frånluftsfläkt
	ST_OP:REAL;		// Utsignal Till- och frånluftsspjäll
	GP11_PV:REAL;
	GP11_FAULT:BOOL;
	GP12_PV:REAL;
	GP12_FAULT:BOOL;
END_STRUCT
END_TYPE

// ---- DUTs/Custom/Redundancy/RedundancyStatus.TcDUT
TYPE RedundancyStatus :
STRUCT
	ENO :  BOOL; 			// Redundans är aktiverad
	UPPSTART_DONE:BOOL;
	TF_CMD:BOOL;
	TF_V:BOOL;
	TF_OP:REAL;
	TL_GP_PV:REAL;
	FF_CMD:BOOL;
	FF_V:BOOL;
	FF_OP:REAL;
	FL_GP_PV:REAL;
	SERVICEBRYTARE:BOOL;
END_STRUCT
END_TYPE

// ---- DUTs/Custom/SmokeControl/SxDuoInterface.TcDUT
TYPE SxDuoInterface :
STRUCT
	{attribute 'TcEncoding':='UTF-8'}
	TEXT_PV: STRING; // Place identifier
	FIRE_AL: BOOL; // Fire alarm
	DAMPER1_AL: BOOL; // Damper 1 alarm
	EXERCISING_V: BOOL; // Exercising
	DAMPER2_AL: BOOL; // Damper 2 alarm
	DAMPER1_V1: BOOL; // Damper 1 open
	DAMPER1_V0: BOOL; // Damper 1 closed
	DAMPER2_V1: BOOL; // Damper 2 open
	DAMPER2_V0: BOOL; // Damper 2 closed
	FIRE_FAULT: BOOL; // Service alarm
	COMM_FAULT: BOOL; // Communication error
END_STRUCT
END_TYPE

// ---- DUTs/Custom/_Standard/AdsTags.TcDUT
TYPE AdsTags :
STRUCT
	Settings: GreenMasterSettings; // Settings for the GreenMaster unit
	Status: GreenMasterStatus; // Status for the GreenMaster unit
	//Schedule1: TimeChannelSettings := (AllDays := TRUE, EN := TRUE, OffHour := 23, OffMinute := 59); // Operating schedule for the GreenMaster unit
	//Schedule2: TimeChannelSettings; // Operating schedule for the GreenMaster unit
	//Schedule3: TimeChannelSettings; // Operating schedule for the GreenMaster unit
	//ScheduleFallback: TimeChannelSettings := (AllDays := TRUE, EN := TRUE, OnHour := 5, OnMinute := 30, OffHour := 20, OffMinute := 00); // Operating schedule for the GreenMaster unit on watchdog trig
END_STRUCT
END_TYPE

// ---- DUTs/Custom/_Standard/GreenMasterSettings.TcDUT
// Settings for GreenMaster
TYPE GreenMasterSettings :
STRUCT
RemoteStart :  INT := 1; //  Remote (WebPort) unit activation (-1=Auto, 0=unit off, 1=normal speed, 2=high speed)
ResetAlarms :  BOOL :=FALSE; //  Reset alarms
VentilationEN: BOOL := TRUE;
TemperatureControlEN: BOOL := TRUE;

TX1_EFF_AD :  TIME :=T#5M; //  Alarm delay low efficiency (s) |||| Larmfördröjning låg verkningsgrad (s) $(unit "s")
TX1_EFF_ALL :  REAL :=0.3; //  Alarm limit low efficiencyLimit |||| Larmgräns låg verkninggrad $(unit "%")

T_BT1_AD: TIME := T#10M; //  Alarm delay temperature deviation (s) |||| Larmfördröjning temperatur-avvikelse (s) $(unit "s")
T_BT1_ADL: REAL := 4; //  Alarm limit temperature deviation |||| Larmgräns temperatur-avvikelse $(unit "°C")
T_GQ1_AD: TIME := T#5S; //  Alarm delay supply fan (s) |||| Larmfördröjning tilluftsfläkt (s) $(unit "s")
F_GQ1_AD: TIME := T#5S; //  Alarm delay extract fan (s) |||| Larmfördröjning frånluftsfläkt (s) $(unit "s")
T_BP2_AD: TIME := T#5S; //  Alarm delay high pressure (s) |||| Larmfördröjning högt tryck (s) $(unit "s")
T_BP2_AHL: REAL := 150; //  Alarm limit high pressure |||| Larmgräns högt tryck $(unit "Pa")
F_BP2_AD: TIME := T#5S; //  Alarm delay high pressure (s) |||| Larmfördröjning högt tryck (s) $(unit "s")
F_BP2_AHL: REAL := 150; //  Alarm limit high pressure |||| Larmgräns högt tryck $(unit "Pa")
F_QM2_SP1: INT:= 48;//  Exercise interval F.QM2 (hour) |||| Motioneringsintervall F.QM2 (timma) $(unit "hour")
F_QM2_SP2: INT:= 10;//  Exercise start hour F.QM2 (hour) |||| Motionering F.QM2 starttimma (timma) $(unit "hour")
F_QM2_SP3: INT:= 30;//  Exercise start minute F.QM2 (minute) |||| Motionering F.QM2 startminut (minuter) $(unit "minute")
EXT_QM_SP1: INT:= 48;//  Exercise interval external dampers (hour) |||| Motioneringsintervall externa spjäll (timma) $(unit "hour")
EXT_QM_SP2: INT:= 10;//  Exercise start hour external dampers (hour) |||| Motionering externa spjäll starttimma (timma) $(unit "hour")
EXT_QM_SP3: INT:= 30;//  Exercise start minute external dampers (minute) |||| Motionering externa spjäll startminut (minut) $(unit "minute")
T_BP1_AD: TIME := T#10M; //  Alarm delay supply pressure deviation (s) |||| Larmfördröjning avvikelse tilluftstryck (s) $(unit "s")
T_BP1_ADL: REAL := 30; //  Alarm limit supply pressure deviation |||| Larmgräns avvikelse tilluftstryck $(unit "Pa")
F_BP1_AD: TIME := T#10M; //  Alarm delay extract pressure deviation (s) |||| Larmfördröjning avvikelse frånluftstryck (s) $(unit "s")
F_BP1_ADL: REAL := 30; //  Alarm limit extract pressure deviation |||| Larmgräns avvikelse frånluftstryck $(unit "Pa")

Temperature_SP :  LREAL :=20; //  Temperature Set Point, C
TemperatureControlPV :  INT :=0; //  0 = Use T.BT1, 1 = Use F.BT1
//SetPointOffsetCurve :  SetPointOffsetCurve := (Y1 := 20, Y2 := 20, Y3 := 20, Y4 := 20, Y5 := 20, Y6 := 20, Y7 := 20, Y8 := 20, Y9 := 20); // Outdoorcompensation temperature
T_BT1_CURVE :  SetPointOffsetCurve; // Outdoorcompensation temperature

TemperatureControl_P :  REAL :=10; //  Temperature control P
TemperatureControl_I :  TIME :=T#2M; //  Temperature control I (s) $(unit "s")
TemperatureControl_D :  TIME :=T#0M; //  Temperature control D (s) $(unit "s")
StartupHeatRecoveryTime :  TIME :=T#0M; //  Time at startup to recover (s) $(unit "s")
PostFireVentilationTime :  TIME :=T#1M; //  Time to ventilate when returning to operation after fire alarm (s) $(unit "s")
SupplyFanControlMode :  FanControlTypes ; //  Control mode (0=Pressure/T.BP1, 1=Flow/T.BF1) for Supply Air
SupplyFan_SP :  REAL :=0 ; //  Supply air control Set Point
SupplyFanHighSpeed_SP :  REAL ; //  Supply air control high speed Set Point
//SupplyFanOffsetCurve :  SetPointOffsetCurve := (Y1 := 165, Y2 := 165, Y3 := 165, Y4 := 165, Y5 := 165, Y6 := 165, Y7 := 165, Y8 := 165, Y9 := 165); // Outdoorcompensation temperature
F_GQ1_CURVE:  SetPointOffsetCurve; // Outdoorcompensation temperature

SupplyFanControl_P :  REAL :=2; //  Supply air control P
SupplyFanControl_I :  TIME :=T#2M; //  Supply air control I $(unit "s")
ExtractFanControlMode :  FanControlTypes ; //  Control mode (0=Pressure/F.BP1, 1=Flow/F.BF1) for Extract Air
ExtractFan_SP :  REAL := 0; //  Extract air control Set Point
ExtractFanHighSpeed_SP :  REAL ; //  Extract air control high speed Set Point
//ExtractFanOffsetCurve :  SetPointOffsetCurve := (Y1 := 160, Y2 := 160, Y3 := 160, Y4 := 160, Y5 := 160, Y6 := 160, Y7 := 160, Y8 := 160, Y9 := 160); // Outdoorcompensation temperature
T_GQ1_CURVE :  SetPointOffsetCurve; // Outdoorcompensation temperature

ExtractFanControl_P :  REAL :=2; //  Extract air control P
ExtractFanControl_I :  TIME :=T#2M; //  Extract air control I $(unit "s")
NightCoolingEN :  BOOL :=FALSE; //  Use Night cooling
NightCoolingTemperatureSP :  REAL :=18.0; //  Night cooling temperature Set Point, C
FanStopDelayTime :  TIME :=T#2M; //  Fan stop delay cool down period $(unit "s")
WatchdogEnabled :  BOOL :=FALSE; //  Watchdog enable - enables unit on watchdog update failure 
Watchdog :  INT :=0; //  Watchdog counter to be changed at a minimum every 5 minutes (when enabled)  
TX1_M :  BOOL; // Heat exchanger manual override
T_GQ1_M :  BOOL; //  Supply air fan control manual override
F_GQ1_M :  BOOL; //  Extract air fan control manual override
C_QN1_M :  BOOL; //  Cool supply control valve manual override
H_QN1_M :  BOOL; //  Heat supply control valve manual override
TX1_OPM :  REAL; //  Heat exchanger manual value $(scale "0 1 0 100", unit "%")
T_GQ1_OPM :  REAL; //  Supply air fan control manual value $(scale "0 1 0 100", unit "%")
F_GQ1_OPM :  REAL; //  Extract air fan control manual value $(scale "0 1 0 100", unit "%")
C_QN1_OPM :  REAL; //  Cool supply control valve manual value $(scale "0 1 0 100", unit "%")
H_QN1_OPM :  REAL; //  Heat supply control valve manual value $(scale "0 1 0 100", unit "%")

TC: TimeChannel_CT_CF;

FREEZE_ALL: REAL := 4; // Freeze protection alarm level$(unit "%C)

// Manual mode
H_GP1_M :  BOOL; // Manöver pump värme
C_GP1_M :  BOOL; // Manöver pump kyla
F_QM1_M :  BOOL; // Frånluftsspjäll manöver
T_QM1_1_M :  BOOL; // Sektionsavfrostningsspjäll 1 manöver
T_QM1_2_M :  BOOL; // Sektionsavfrostningsspjäll 2 manöver
T_QM1_3_M :  BOOL; // Sektionsavfrostningsspjäll 3 manöver
T_QM1_4_M :  BOOL; // Sektionsavfrostningsspjäll 4 manöver
T_QM1_5_M :  BOOL; // Sektionsavfrostningsspjäll 5 manöver
T_QM1_6_M :  BOOL; // Sektionsavfrostningsspjäll 6 manöver
F_QM2_M :  BOOL; // Brandförbigångsspjäll (FID) manöver
T_QM2_M :  BOOL; // spjäll manöver
T_QM3_M :  BOOL; // spjäll manöver

// Manual command
H_GP1_MCMD :  BOOL; // Manöver pump värme
C_GP1_MCMD :  BOOL; // Manöver pump kyla
F_QM1_MCMD :  BOOL; // Frånluftsspjäll manöver
T_QM1_1_MCMD :  BOOL; // Sektionsavfrostningsspjäll 1 manöver
T_QM1_2_MCMD :  BOOL; // Sektionsavfrostningsspjäll 2 manöver
T_QM1_3_MCMD :  BOOL; // Sektionsavfrostningsspjäll 3 manöver
T_QM1_4_MCMD :  BOOL; // Sektionsavfrostningsspjäll 4 manöver
T_QM1_5_MCMD :  BOOL; // Sektionsavfrostningsspjäll 5 manöver
T_QM1_6_MCMD :  BOOL; // Sektionsavfrostningsspjäll 6 manöver
F_QM2_MCMD :  BOOL; // Brandförbigångsspjäll (FID) manöver
T_QM2_MCMD :  BOOL; // spjäll manöver
T_QM3_MCMD :  BOOL; // spjäll manöver

END_STRUCT
END_TYPE

// ---- DUTs/Custom/_Standard/GreenMasterStatus.TcDUT
TYPE GreenMasterStatus :
STRUCT
ENO :  BOOL; // Unit is operating |||| Aggregatet är i drift
AUTO :  BOOL; // Aggregatet är i auto
HAND :  BOOL; // Aggregatet är i hand
SFP_PV: REAL; // Current SFPv |||| Aktuellt SFPv $(scale "0 5 0 5", unit "kW/(m³s)", format "0.000")
TX1_EFF_LAL: BOOL; // Larm låg verkningsgrad
MODE_PV1 : INT; // Driftmod 0=stopp, 1=halvfart, 2=helfart
F_BR1_AL :  BOOL; // Brandlarm F.BR1
TC_V : BOOL; // Tidkanal i aggregat är aktiv
F_BR1_FAULT :  BOOL; // Servicelarm F.BR1
FIRE_AL :  BOOL; // Brandlarm
F_BRT2_AL :  BOOL; // Brandlarm frånluft temperatur (normalt 45 C)
F_BRT3_AL :  BOOL; // Brandlarm frånluft temperatur och tryck (normalt 38 C och 170 Pa)
FUSE_AL :  BOOL; // Utlöst säkring
T_BR1_AL :  BOOL; // Brandlarm T.BR1
T_BR1_FAULT :  BOOL; // Servicelarm T.BR1
T_GQ1_AL :  BOOL; // Driftfel tilluftsfläkt
F_GQ1_AL :  BOOL; // Driftfel frånluftsfläkt
H_GP1_V :  BOOL; // Driftindikering pump värme
H_GP1_AL :  BOOL; // Driftfel pump värme
C_GP1_V :  BOOL; // Driftindikering pump kyla
C_GP1_AL :  BOOL; // Driftfel pump kyla
T_GQ_AL1 :  BOOL; // Tilluftsfläkt handstartad
T_GQ_AL2 :  BOOL; // Tilluftsfläkt handstoppad
F_GQ_AL1 :  BOOL; // Frånluftsfläkt handstartad
F_GQ_AL2 :  BOOL; // Frånluftsfläkt handstoppad
QM_AL :  BOOL; // Brandspjäll i fel läge
TX1_EFF_PV :  REAL; // Verkningsgrad VVX $(scale "0 1 0 100", unit "%")
H_GP1_CMD :  BOOL; // Manöver pump värme
C_GP1_CMD :  BOOL; // Manöver pump kyla
F_QM1_CMD :  BOOL; // Frånluftsspjäll manöver
T_QM1_CMD :  BOOL; // Tilluftsspjäll manöver
T_QM1_1_CMD :  BOOL; // Sektionsavfrostningsspjäll 1 manöver
T_QM1_2_CMD :  BOOL; // Sektionsavfrostningsspjäll 2 manöver
T_QM1_3_CMD :  BOOL; // Sektionsavfrostningsspjäll 3 manöver
T_QM1_4_CMD :  BOOL; // Sektionsavfrostningsspjäll 4 manöver
T_QM1_5_CMD :  BOOL; // Sektionsavfrostningsspjäll 5 manöver
T_QM1_6_CMD :  BOOL; // Sektionsavfrostningsspjäll 6 manöver
F_QM2_CMD :  BOOL; // Brandförbigångsspjäll (FID) manöver
F_QM2_V0 :  BOOL; // Brandförbigångsspjäll (FID) stängt
F_QM2_V1 :  BOOL; // Brandförbigångsspjäll (FID) öppet
TEMPERATURE_CSP : REAL; // Aktuellt börvärdetemperatur
T_BT2_PV :  REAL; // Utetemperatur (aggregat)
T_BT2_FAULT :  BOOL; // Utetemperatur (aggregat) givarfel
T_BT3_PV :  REAL; // Tilluftstemperatur före efterbehandling (aggregat)
T_BT3_FAULT :  BOOL; // Tilluftstemperatur före efterbehandling (aggregat) givarfel
H_BT1_PV :  REAL; // Frysskyddstemperatur (batteri)
H_BT1_FAULT :  BOOL; // Frysskyddstemperatur (batteri) givarfel
H_BT1_LAL :  BOOL; // Frysskyddslarm
BT1_PV :  REAL; // Utomhustemperatur (fasad)
BT1_FAULT :  BOOL; // Utomhustemperatur (fasad) givarfel
F_BT2_PV :  REAL; // Avluftstemperatur (aggregat)
F_BT2_FAULT :  BOOL; // Avluftstemperatur (aggregat) givarfel
T_BP2_PV :  REAL; // Differenstryck tilluftsfilter
T_BP2_FAULT :  BOOL; // Differenstryck tilluftsfilter givarfel
T_BP2_HAL :  BOOL; // Differenstryck tilluftsfilter Larm
F_BP2_PV :  REAL; // Differenstryck frånluftsfilter
F_BP2_FAULT :  BOOL; // Differenstryck frånluftsfilter givarfel
F_BP2_HAL :  BOOL; // Differenstryck frånluftsfilter Larm
F_BP3_PV :  REAL; // Differenstryck VVX
F_BP3_FAULT :  BOOL; // Differenstryck VVX givarfel
F_BP3_AL :  BOOL; // Differenstryck VVX Larm
T_GQ1_OP :  REAL; // Utsignal tilluftsfläkt $(scale "0 1 0 100", unit "%")
F_GQ1_OP :  REAL; // Utsignal frånluftsfläkt $(scale "0 1 0 100", unit "%")
T_GQ1_V :  BOOL; // Drift tilluftsfläkt
F_GQ1_V :  BOOL; // Drift frånluftsfläkt
TX1_OP :  REAL; // Utsignal VVX $(scale "0 1 0 100", unit "%")
H_QN1_OP :  REAL; // Utsignal värmeventil $(scale "0 1 0 100", unit "%")
C_QN1_OP :  REAL; // Utsignal kylventil $(scale "0 1 0 100", unit "%")
T_QM2_CMD :  BOOL; // spjäll manöver
T_QM2_V0 :  BOOL; // Brandförbigångsspjäll (FID) stängt
T_QM2_V1 :  BOOL; // Brandförbigångsspjäll (FID) öppet
T_QM3_CMD :  BOOL; // spjäll manöver
T_QM3_V0 :  BOOL; // Brandförbigångsspjäll (FID) stängt
T_QM3_V1 :  BOOL; // Brandförbigångsspjäll (FID) öppet

F_BT1_PV :  REAL; // Frånluftstemperatur (aggregat)
F_BT1_FAULT :  BOOL; // Frånluftstemperatur (aggregat) givarfel
F_BT1_AL :  BOOL; // Frånluftstemperatur (aggregat) Larm
T_BT1_PV :  REAL; // Tilluftstemperatur (kanal)
T_BT1_FAULT :  BOOL; // Tilluftstemperatur (kanal) givarfel
T_BT1_AL :  BOOL; // Tilluftstemperatur (kanal) Larm
BT2_PV :  REAL; // Inomhustemperatur (vägg)
BT2_FAULT :  BOOL; // Inomhustemperatur (vägg) givarfel
BT2_AL :  BOOL; // Inomhustemperatur (vägg) Larm

T_BF1_PV :  REAL; // Tilluftsflöde
T_BF1_CSP : REAL; // Beräknat börvärde tilluftsflöde
T_BF1_FAULT :  BOOL; // Tilluftsflöde givarfel
T_BF1_AL :  BOOL; // Tilluftsflöde Larm
T_BP1_PV :  REAL; // Tilluftstryck
T_BP1_CSP : REAL; // Beräknat börvärde tilluftstryck
T_BP1_FAULT :  BOOL; // Tilluftstryck givarfel
T_BP1_AL :  BOOL; // Tilluftstryck Larm

F_BF1_PV :  REAL; // Frånluftsflöde
F_BF1_CSP : REAL; // Beräknat börvärde frånluftsflöde
F_BF1_FAULT :  BOOL; // Frånluftsflöde givarfel
F_BF1_AL :  BOOL; // Frånluftsflöde Larm
F_BP1_PV :  REAL; // Frånluftstryck
F_BP1_CSP : REAL;	// Beräknat börvärde frånluftstryck"
F_BP1_FAULT :  BOOL; // Frånluftstryck givarfel
F_BP1_AL :  BOOL; // Frånluftstryck Larm
PLC_VERSION_PV: STRING; // PLC version (major.minor.patch)
TIMEANDDATE_PV: STRING; // Current time in the PLC unit |||| Aktuell tid i PLC-enheten
NightCooling_V :  BOOL; //  Active night time cooling  
TX1_AL: BOOL; // Larm värmeväxlare (rotationsvakt)
TX1_E1: REAL; // Återvunnen energi från värmeväxlare till tilluft (dag)
TX1_E2: REAL; // Återvunnen energi från värmeväxlare till tilluft (senaste dag)
TX1_E3: REAL; // Återvunnen energi från värmeväxlare till tilluft (månad)
TX1_E4: REAL; // Återvunnen energi från värmeväxlare till tilluft (senaste månad)
TX1_E5: REAL; // Återvunnen energi från värmeväxlare till tilluft (år)
TX1_E6: REAL; // Återvunnen energi från värmeväxlare till tilluft (senaste år)
H_BT1_E1: REAL; // Energi från värmebatteri till tilluft (dag)
H_BT1_E2: REAL; // Energi från värmebatteri till tilluft (senaste dag)
H_BT1_E3: REAL; // Energi från värmebatteri till tilluft (månad)
H_BT1_E4: REAL; // Energi från värmebatteri till tilluft (senaste månad)
H_BT1_E5: REAL; // Energi från värmebatteri till tilluft (år)
H_BT1_E6: REAL; // Energi från värmebatteri till tilluft (senaste år)
END_STRUCT
END_TYPE

// ---- DUTs/Custom/_Standard/TimeChannel_CT_CF.TcDUT
TYPE TimeChannel_CT_CF :
STRUCT
	CT1 : UINT ; // Mån Till 1
	CT2 : UINT ; // Tis Till 1
	CT3 : UINT ; // Ons Till 1
	CT4 : UINT ; // Tor Till 1
	CT5 : UINT ; // Fre Till 1
	CT6 : UINT ; // Lör Till 1
	CT7 : UINT ; // Sön Till 1
	
	CT11 : UINT ; // Mån Till 2
	CT12 : UINT ; // Tis Till 2
	CT13 : UINT ; // Ons Till 2
	CT14 : UINT ; // Tor Till 2
	CT15 : UINT ; // Fre Till 2
	CT16 : UINT ; // Lör Till 2
	CT17 : UINT ; // Sön Till 2
	
	CT21 : UINT ; // Mån Till 3
	CT22 : UINT ; // Tis Till 3
	CT23 : UINT ; // Ons Till 3
	CT24 : UINT ; // Tor Till 3
	CT25 : UINT ; // Fre Till 3
	CT26 : UINT ; // Lör Till 3
	CT27 : UINT ; // Sön Till 3
	
	CF1 : UINT := 2400; // Mån Från 1
	CF2 : UINT := 2400; // Tis Från 1
	CF3 : UINT := 2400; // Ons Från 1
	CF4 : UINT := 2400; // Tor Från 1
	CF5 : UINT := 2400; // Fre Från 1
	CF6 : UINT := 2400; // Lör Från 1
	CF7 : UINT := 2400; // Sön Från 1
	
	CF11 : UINT ; // Mån Från 2
	CF12 : UINT ; // Tis Från 2
	CF13 : UINT ; // Ons Från 2
	CF14 : UINT ; // Tor Från 2
	CF15 : UINT ; // Fre Från 2
	CF16 : UINT ; // Lör Från 2
	CF17 : UINT ; // Sön Från 2
	
	CF21 : UINT ; // Mån Från 3
	CF22 : UINT ; // Tis Från 3
	CF23 : UINT ; // Ons Från 3
	CF24 : UINT ; // Tor Från 3
	CF25 : UINT ; // Fre Från 3
	CF26 : UINT ; // Lör Från 3
	CF27 : UINT ; // Sön Från 3

END_STRUCT
END_TYPE

// ---- DUTs/Defrost/DefrostSections.TcDUT
{attribute 'qualified_only'}
{attribute 'strict'}
TYPE DefrostSections :
(
	S0 := 0, S1, S2, S3, S4, S5, S6, S1_3, S2_4, S3_5, S4_6, S1_3_5, S2_4_6
);
END_TYPE

// ---- DUTs/GreenMaster/SystemStatesRunMode.TcDUT
{attribute 'qualified_only'}
{attribute 'strict'}
TYPE SystemStatesRunMode :
(
	Off := 0, LowSpeed, HighSpeed
);
END_TYPE

// ---- DUTs/GreenMaster/SystemStatesRunModeExternal.TcDUT
{attribute 'qualified_only'}
{attribute 'strict'}
TYPE SystemStatesRunModeExternal :
(
	Auto := -1, Stop, LowSpeed, HighSpeed
);
END_TYPE

// ---- DUTs/IO/AI3468.TcDUT
TYPE AI3468 :
STRUCT
	AI1 AT %I*: INT;
	AI1_Error AT %I*: BOOL;
	AI2 AT %I*: INT;
	AI2_Error AT %I*: BOOL;
END_STRUCT
END_TYPE

// ---- DUTs/Parameters/Alarm/AlarmControl.TcDUT
TYPE AlarmControl :
STRUCT
	ResetAlarms: BOOL;
END_STRUCT
END_TYPE

// ---- DUTs/Parameters/Alarm/AlarmDelays.TcDUT
// MUST be in same order and number as AlarmSignals
TYPE AlarmDelays :
STRUCT
	A: AlarmsDelaysA;
	B: AlarmsDelaysB;
	C: AlarmsDelaysC;
END_STRUCT
END_TYPE

// ---- DUTs/Parameters/Alarm/AlarmLimits.TcDUT
TYPE AlarmLimits :
STRUCT
	FireAlarmExtractAir: LREAL := 38; // $(W1,S,R0)
	RegulationDeviationAlarm: LREAL := 2; // $(W1,S,R0)
	SupplyAirPressureDeviationAlarm: LREAL := 30; // $(W1,S,R0)
	ExtractAirPressureDeviationAlarm: LREAL := 30; // $(W1,S,R0)
	SupplyAirFlowDeviationAlarm: LREAL := 0.3; // $(W1,S,R0)
	ExtractAirFlowDeviationAlarm: LREAL := 0.3; // $(W1,S,R0)
	HeatExchangerEfficiencyAlarm: LREAL; // $(W1,S,R0)
	DefrostAlarm: LREAL := -1; // $(W1,S,R0)
	SupplyFilterAlarm: LREAL := 150; // $(W1,S,R0)
	ExtractFilterAlarm: LREAL := 150; // $(W1,S,R0)
END_STRUCT
END_TYPE

// ---- DUTs/Parameters/Alarm/AlarmLimitsA.TcDUT
TYPE AlarmLimitsA :
STRUCT
	FireExtractTemperature: REAL := 45;
	FireExtractPressureTemperature: REAL := 38;
	FireExtractPressure: REAL := 170;
	Freeze: REAL := 8;
END_STRUCT
END_TYPE

// ---- DUTs/Parameters/Alarm/AlarmLimitsB.TcDUT
TYPE AlarmLimitsB :
STRUCT
	RegulationDeviation: REAL := 4;
	SupplyAirPressureDeviation: REAL := 30;
	ExtractAirPressureDeviation: REAL := 30;
	SupplyAirFlowDeviation: REAL := 0.3;
	ExtractAirFlowDeviation: REAL := 0.3;
	HeatExchangerEfficiency: REAL := 0.3; // $(scale "0 1 0 100", unit "%")
	Defrost: REAL := -1;
	SupplyFilter: REAL := 150;
	ExtractFilter: REAL := 150;
	HeatExchangerHighPressure: REAL := 310;
	OperatingTime: LTIME := LTIME#15H;
END_STRUCT
END_TYPE

// ---- DUTs/Parameters/Alarm/AlarmLimitsC.TcDUT
TYPE AlarmLimitsC :
STRUCT
END_STRUCT
END_TYPE

// ---- DUTs/Parameters/Alarm/AlarmParameters.TcDUT
TYPE AlarmParameters :
STRUCT
	Control: AlarmControl;
	Enabled: AlarmSignals := ( 	A := ( 		
										FireExtract := TRUE,
										FireExtractTemperature := TRUE,
										FireExtractPressure := TRUE,
										FireExtractExternal := TRUE,
										FireLocal := TRUE,
										FireSupply := TRUE,
										Freeze := TRUE,
										Fuse := TRUE,
										Cold := TRUE,
										Aux := TRUE
									),
									B := (	
										RegulationDeviation := TRUE,
										SupplyAirDeviation := TRUE,
										ExtractAirDeviation := TRUE,
										SupplyFan := TRUE,
										ExtractFan := TRUE,
										HeatExchangerEfficiency := TRUE,
										Defrost := TRUE,
										SupplyFilter := TRUE,
										ExtractFilter := TRUE,
										SmokeDetectorServiceSupply := TRUE,
										SmokeDetectorServiceExtract := TRUE,
										Pump1 := TRUE,
										DamperError := TRUE,
										CommunicationError := TRUE,
										DamperModuleService := TRUE,
										TX1Fail := TRUE
									),
									C := (	
										ExternalSmokeControl := TRUE,
										ModbusRTU := TRUE,
										ModbusTCP := TRUE,
										SensorFailure := TRUE
									));
	AutoReset: AlarmSignals := ( 	A := ( 	FirePanelSupplyStart := TRUE,  
											FirePanelSupplyStop := TRUE, 
											FirePanelExtractStart := TRUE, 
											FirePanelExtractStop := TRUE,
											Fuse := TRUE,
											FireExtract := FALSE,
											FireExtractTemperature := FALSE,
											FireExtractPressure := FALSE,
											FireExtractExternal := FALSE,
											FireLocal := FALSE,
											FireSupply := TRUE,
											AL01 := TRUE,
											AL02 := TRUE,
											AL03 := TRUE,
											AL04 := TRUE,
											AL05 := TRUE,
											AL06 := TRUE,
											AL07 := TRUE,
											AL08 := TRUE
									),
									B := (	RegulationDeviation := TRUE,
											SupplyAirDeviation := TRUE,
											ExtractAirDeviation := TRUE,
											SupplyFan := FALSE,
											ExtractFan := FALSE,
											HeatExchangerEfficiency := TRUE,
											Defrost := TRUE,
											SupplyFilter := TRUE,
											ExtractFilter := TRUE,
											SmokeDetectorServiceSupply := TRUE,
											Pump1 := TRUE,
											Pump2 := TRUE,
											CommunicationError := TRUE,
											TX1Fail := TRUE
									),
									C := (	ExternalSmokeControl := TRUE,
											ModbusRTU := TRUE,
											ModbusTCP := TRUE,
											SensorFailure := TRUE
									));
	Limits: AlarmLimits;
	Delay: AlarmDelays; // MUST be in same order and number as AlarmSignals
	Polarity: AlarmSignals := ( A:= ( FireExtract := FALSE ));
	Active: AlarmSignals;
	Status: AlarmSignals;	
	
END_STRUCT
END_TYPE

// ---- DUTs/Parameters/Alarm/AlarmsA.TcDUT
TYPE AlarmsA :
STRUCT
	FireExtract: BOOL;
	FireExtractTemperature: BOOL;
	FireExtractPressure: BOOL;
	FireExtractExternal: BOOL;
	FireLocal: BOOL;
	FireSupply: BOOL;
	FreezeGuard: BOOL;
	Fuse: BOOL;
	Cold: BOOL;
	Aux: BOOL;
	FirePanelSupplyStart: BOOL;
	FirePanelSupplyStop: BOOL;
	FirePanelExtractStart: BOOL;
	FirePanelExtractStop: BOOL;
	AL01: BOOL;
	AL02: BOOL;
	AL03: BOOL;
	AL04: BOOL;
	AL05: BOOL;
	AL06: BOOL;
	AL07: BOOL;
	AL08: BOOL;
	SupplyDamperError: BOOL;
	ExtractDamperError: BOOL;
END_STRUCT
END_TYPE

// ---- DUTs/Parameters/Alarm/AlarmsB.TcDUT
TYPE AlarmsB :
STRUCT
	RegulationDeviation: BOOL;
	SupplyAirDeviation: BOOL;
	ExtractAirDeviation: BOOL;
	SupplyFan: BOOL;
	ExtractFan: BOOL;
	HeatExchangerEfficiency: BOOL;
	Defrost: BOOL;
	SupplyFilter: BOOL;
	ExtractFilter: BOOL;
	SmokeDetectorServiceSupply: BOOL;
	SmokeDetectorServiceExtract: BOOL;
	Pump1: BOOL;
	Pump2: BOOL;
	DamperError: BOOL;
	CommunicationError: BOOL;
	DamperModuleService: BOOL;
	Tx1Fail: BOOL;
END_STRUCT
END_TYPE

// ---- DUTs/Parameters/Alarm/AlarmsC.TcDUT
TYPE AlarmsC :
STRUCT
	ExternalSmokeControl: BOOL;
	ModbusRTU: BOOL;
	ModbusTCP: BOOL;
	SensorFailure: BOOL;
END_STRUCT
END_TYPE

// ---- DUTs/Parameters/Alarm/AlarmsDelaysA.TcDUT
// MUST be in same order and number as AlarmSignals
TYPE AlarmsDelaysA :
STRUCT
	FireExtract: TIME := T#5S;
	FireExtractTemperature: TIME := T#5S;
	FireExtractPressure: TIME := T#5S;
	FireExtractExternal: TIME := T#5S;
	FireLocal: TIME := T#5S;
	FireSupply: TIME := T#5S;
	Freeze: TIME := T#5S;
	Fuse: TIME := T#5S;
	Cold: TIME := T#5S;
	Aux: TIME := T#5S;
	FirePanelSupplyStart: TIME := T#1S;
	FirePanelSupplyStop: TIME := T#1S;
	FirePanelExtractStart: TIME := T#1S;
	FirePanelExtractStop: TIME := T#1S;
	AL01: TIME := T#5S;
	AL02: TIME := T#5S;
	AL03: TIME := T#5S;
	AL04: TIME := T#5S;
	AL05: TIME := T#5S;
	AL06: TIME := T#5S;
	AL07: TIME := T#5S;
	AL08: TIME := T#5S;
	SupplyDamperError: TIME := T#5S;
	ExtractDamperError: TIME := T#5S;
END_STRUCT
END_TYPE

// ---- DUTs/Parameters/Alarm/AlarmsDelaysB.TcDUT
// MUST be in same order and number as AlarmSignals
TYPE AlarmsDelaysB :
STRUCT
	RegulationDeviation: TIME := T#60M;
	SupplyAirDeviation: TIME := T#60M;
	ExtractAirDeviation: TIME := T#60M;
	SupplyFan: TIME := T#60S;
	ExtractFan: TIME := T#60S;
	HeatExchangerEfficiency: TIME := T#1H;
	Defrost: TIME := T#5S;
	SupplyFilter: TIME := T#1H;
	ExtractFilter: TIME := T#1H;
	SmokeDetectorServiceSupply: TIME := T#5S;
	SmokeDetectorServiceExtract: TIME := T#5S;
	Pump1: TIME := T#5S;
	Pump2: TIME := T#5S;
	DamperError: TIME := T#30S;
	CommunicationError: TIME := T#30S;
	DamperModuleService: TIME := T#5S;
	Tx1Fail: TIME := T#1M;
END_STRUCT
END_TYPE

// ---- DUTs/Parameters/Alarm/AlarmsDelaysC.TcDUT
// MUST be in same order and number as AlarmSignals
TYPE AlarmsDelaysC :
STRUCT
	ExternalSmokeControl: TIME := T#5S;
	ModbusRTU: TIME := T#5S;
	ModbusTCP: TIME := T#5S;
	SensorFailure: TIME := T#5S;
END_STRUCT
END_TYPE

// ---- DUTs/Parameters/Alarm/AlarmSignals.TcDUT
TYPE AlarmSignals :
STRUCT
	A: AlarmsA;
	B: AlarmsB;
	C: AlarmsC;
END_STRUCT
END_TYPE

// ---- DUTs/Alarms/AlarmLog.TcDUT
TYPE AlarmLog :
STRUCT
	Head: INT;
	Tail: INT;
	Alarms: ARRAY [Globals.AlarmsLow..Globals.AlarmsHigh] OF AlarmEvent;
END_STRUCT
END_TYPE

// ---- DUTs/Alarms/AlarmEvent.TcDUT
TYPE AlarmEvent :
STRUCT
	TimeStamp: DT;
	Signals: AlarmSignals; 
	Status: AlarmSignals; 
	Acknowledged: BOOL;
	AcknowledgedTime: DT;
	{attribute 'TcEncoding':='UTF-8'}
	AcknowledgedBy: STRING(20);
	Reset: BOOL;
	ResetTime: DT;
	{attribute 'TcEncoding':='UTF-8'}
	ResetBy: STRING(20);
	{attribute 'TcEncoding':='UTF-8'}
	Message: STRING(20);
	{attribute 'TcEncoding':='UTF-8'}
	Notes: STRING(20);
	{attribute 'TcEncoding':='UTF-8'}
	JSON: BOOL;
END_STRUCT
END_TYPE

// ---- DUTs/Defrost/DefrostStates.TcDUT
{attribute 'qualified_only'}
{attribute 'strict'}
TYPE DefrostStates :
(
	Normal := 0, ReducedTF, DualSections, ClosedTF 
);
END_TYPE

// ---- DUTs/Events/Event.TcDUT
TYPE Event :
STRUCT
	Code: INT;
	TimeStamp: DT;
	Kind: EventTypes;
	{attribute 'TcEncoding':='UTF-8'}
	Message: STRING(200);
	{attribute 'TcEncoding':='UTF-8'}
	JSON: BOOL;
END_STRUCT
END_TYPE

// ---- DUTs/Events/EventLogData.TcDUT
TYPE EventLogData :
STRUCT
	Head: INT;
	Tail: INT;
	Events: ARRAY [Globals.EventsLow..Globals.EventsHigh] OF Event;
END_STRUCT
END_TYPE

// ---- DUTs/Events/EventTypes.TcDUT
{attribute 'qualified_only'}
{attribute 'strict'}
TYPE EventTypes :
(
	Verbose := 0, Debug, Information, Warning, Error, Critical
);
END_TYPE

// ---- DUTs/Fans/FanControlTypes.TcDUT
{attribute 'qualified_only'}
{attribute 'strict'}
TYPE FanControlTypes :
(
	Pressure := 0, // Pressure control 
	Flow, // Flow control
	SlaveFlow, // Slave flow control
	Const // Constant setting control
);
END_TYPE

// ---- DUTs/GreenMaster/SystemStates.TcDUT
{attribute 'qualified_only'}
{attribute 'strict'}
{attribute 'to_string'}
TYPE SystemStates :
(
	None := 0, Start, Idle, OpenDampers, StartupHeatRecovery, Run, PostRun, FireHandling, FireHandlingExit, FireExhaust, FireSupply, Ventilate, Exercise
);
END_TYPE

// ---- DUTs/IO/TIoKind.TcDUT
{attribute 'qualified_only'}
{attribute 'strict'}
TYPE TIoKind :
(
	DigitalIn := 0, DigitalOut, AnalogIn, AnalogOut
);
END_TYPE

// ---- DUTs/ModbusRTU/ModbusRegisterType.TcDUT
{attribute 'qualified_only'}
{attribute 'strict'}
TYPE ModbusRegisterType :
(
	InputRegister := 0, HoldingRegister
);
END_TYPE

// ---- DUTs/Parameters/GreenMasterBaseParameters.TcDUT
TYPE GreenMasterBaseParameters :
STRUCT
	System: SystemParameters;
	Regulation: RegulationParameters;
	Alarm: AlarmParameters;
	IO: IoParameters;
	Simulation: SimulationParameters;
END_STRUCT
END_TYPE

// ---- DUTs/Parameters/GreenMasterParametersXXL.TcDUT
TYPE GreenMasterParametersXXL :
STRUCT
	System: SystemParametersXXL;
END_STRUCT
END_TYPE

// ---- DUTs/Parameters/GreenMasterParametersXXLFB.TcDUT
TYPE GreenMasterParametersXXLFB:
STRUCT
END_STRUCT
END_TYPE

// ---- DUTs/Parameters/IO/AnalogInputParameters.TcDUT
TYPE AnalogInputParameters :
STRUCT
	F_BT1: LREAL; // Frånluftstemperatur $(unit "°C")  
    T_BT2: LREAL; // Uteluftstemperatur $(unit "°C")
    T_BT3: LREAL; // Tilluftstemperatur (innan efterbehandling) $(unit "°C")
    H_BT1: LREAL; // Frysskyddstemperatur (används bara om värmebatteri (av vätsketyp) är installerat) $(unit "°C")
    T_BT1: LREAL; // Tilluftstemperatur (efter efterbehandling) $(unit "°C") 
    BT1: LREAL; // Utomhustemperatur (extern utegivare, T.BT2 används som utegivare som standard) $(unit "°C")
    BT2: LREAL; // Rumstemperatur (lokalgivare, används inte i bostadsaggregat) $(unit "°C")
    F_BT2: LREAL; // Avluftstemperatur (tillval) $(unit "°C")
	
    F_BP1: LREAL; // Tryckgivare Frånluftskanal $(unit "Pa")
    T_BP1: LREAL; // Tryckgivare Tilluftskanal $(unit "Pa")
    F_BP2: LREAL; // Tryckgivare Frånluftsfilter $(unit "Pa")
    T_BP2: LREAL; //  Tryckgivare uteluftsfilter $(unit "Pa")
    F_BP3: LREAL; // Tryckgivare VVX $(unit "Pa")
    T_BF1: LREAL; // Flödesgivare Tilluftsfläkt $(unit "m³/h")
    F_BF1: LREAL; // Flödesgivare Frånluftsfläkt $(unit "m³/h")	

	F_BT1_Error: BOOL; 
    T_BT2_Error: BOOL;
    T_BT3_Error: BOOL;
    H_BT1_Error: BOOL;
    T_BT1_Error: BOOL; 
    BT1_Error: BOOL;
    BT2_Error: BOOL;
    F_BT2_Error: BOOL;
	
    F_BP1_Error: BOOL;
    T_BP1_Error: BOOL;
    F_BP2_Error: BOOL;
    T_BP2_Error: BOOL;
    F_BP3_Error: BOOL;
    T_BF1_Error: BOOL;
    F_BF1_Error: BOOL;	

	F_BT1_EN: BOOL := TRUE; 
    T_BT2_EN: BOOL := TRUE;
    T_BT3_EN: BOOL := TRUE;
    H_BT1_EN: BOOL := TRUE;
    T_BT1_EN: BOOL := TRUE; 
    BT1_EN: BOOL := FALSE;
    BT2_EN: BOOL := FALSE;
    F_BT2_EN: BOOL := TRUE;
	
    F_BP1_EN: BOOL := TRUE;
    T_BP1_EN: BOOL := TRUE;
    F_BP2_EN: BOOL := TRUE;
    T_BP2_EN: BOOL := TRUE;
    F_BP3_EN: BOOL := TRUE;
    T_BF1_EN: BOOL := TRUE;
    F_BF1_EN: BOOL := TRUE;	
END_STRUCT
END_TYPE

// ---- DUTs/Parameters/IO/AnalogOutputCalibration.TcDUT
TYPE AnalogOutputCalibration :
STRUCT
	F_QN1: AnalogOutputCalibrationParameters;
	T_GQ1: AnalogOutputCalibrationParameters;
	F_GQ1: AnalogOutputCalibrationParameters;
	C_QN1: AnalogOutputCalibrationParameters := (InvertedOutput := TRUE);
	H_QN1: AnalogOutputCalibrationParameters;
END_STRUCT
END_TYPE

// ---- DUTs/Parameters/IO/AnalogOutputCalibrationParameters.TcDUT
TYPE AnalogOutputCalibrationParameters :
STRUCT
	Output: LREAL;
	Gain: LREAL := 1.0;
	ManualControl: BOOL;
	InvertedOutput: BOOL;
END_STRUCT
END_TYPE

// ---- DUTs/Parameters/IO/AnalogOutputOverrideParameters.TcDUT
TYPE AnalogOutputOverrideParameters :
STRUCT
	F_QN1_Override: BOOL; // VVX-reglering (0-10 V spjäll)
	F_QN1_OverrideValue: LREAL; // VVX-reglering (0-10 V spjäll)
	T_GQ1_Override: BOOL; // Tilluftsfläkt
	T_GQ1_OverrideValue: LREAL; // Tilluftsfläkt
	F_GQ1_Override: BOOL; // Frånluftsfläkt
	F_GQ1_OverrideValue: LREAL; // Frånluftsfläkt
	C_QN1_Override: BOOL; // Kylkrets ventil
	C_QN1_OverrideValue: LREAL; // Kylkrets ventil
	H_QN1_Override: BOOL; // Värmekrets ventil
	H_QN1_OverrideValue: LREAL; // Värmekrets ventil
END_STRUCT
END_TYPE

// ---- DUTs/Parameters/IO/AnalogOutputParameters.TcDUT
TYPE AnalogOutputParameters :
STRUCT
	F_QN1: LREAL; // VVX-reglering (0-10 V spjäll) $(scale "0 1 0 100", unit "%")
	T_GQ1: LREAL; // Tilluftsfläkt $(scale "0 1 0 100", unit "%")
	F_GQ1: LREAL; // Frånluftsfläkt $(scale "0 1 0 100", unit "%")
	C_QN1: LREAL; // Kylkrets ventil $(scale "0 1 0 100", unit "%")
	H_QN1: LREAL; // Värmekrets ventil $(scale "0 1 0 100", unit "%")
END_STRUCT
END_TYPE

// ---- DUTs/Parameters/IO/DigitalInputParameters.TcDUT
TYPE DigitalInputParameters :
STRUCT
	Auto: BOOL; // AUTO (Sluten=Aggregat tillåts till drift via överstyrning)
	FireExtractAlarm: BOOL; // Brandlarm (centralt/rökdetektor frånluft)
	FuseAlarm: BOOL; // Utlöst automatsäkring, larm
	Hand: BOOL; // HAND (Sluten=Aggregat i konstant drift)
	T_GQ1_Alarm: BOOL; // Larm T.GQ1 Tilluftsfläkt
	F_GQ1_Alarm: BOOL; // Larm F.GQ1 Frånluftsfläkt
	F_QM2_Closed: BOOL; // F.QM2 brandspjäll ändläge 1 (spjäll stängt/normalläge)
	F_QM2_Open: BOOL; // F.QM2 brandspjäll ändläge 2 (spjäll öppet/brandläge)
	ExtendedOperation: BOOL; // Förlängd drift
	ServiceAlarmCentralAndSmokeExhaustAir: BOOL; // Servicelarm (centralt/rökdetektor frånluft)
	FireSupplyAlarm: BOOL; // Brandlarm (tilluft)
	ServiceAlarmSupplyAir: BOOL; // Servicelarm (tilluft)
	H_GP1_Running: BOOL; // Ingång för pumpdrift, alt. pumplarm H.GP1 (värme)
	H_GP1_Alarm: BOOL;
	C_GP1_Running: BOOL; // Ingång för pumpdrift, alt. pumplarm C.GP1 (kyla)
	C_GP1_Alarm: BOOL;
	TX1_Running: BOOL; // Ingång för rotationsvakt värmeväxlare (TX1)
	ResetAlarm: BOOL; // Larmåterställning
	P2_Running: BOOL;
	ExpansionVesselAlarm: BOOL;
	FirePanelSupplyStart: BOOL;
	FirePanelSupplyStop: BOOL;
	FirePanelExtractStart: BOOL;
	FirePanelExtractStop: BOOL;
END_STRUCT
END_TYPE

// ---- DUTs/Parameters/IO/DigitalOutputOverrideParameters.TcDUT
TYPE DigitalOutputOverrideParameters :
STRUCT
    H_GP1_Override: BOOL; // Cirkulationspump värmekrets
    H_GP1_OverrideValue: BOOL; // Cirkulationspump värmekrets
    C_GP1_Override: BOOL; // Cirkulationspump kylkrets
    C_GP1_OverrideValue: BOOL; // Cirkulationspump kylkrets
    F_QM1_Override: BOOL; // Frånluftsspjäll
    F_QM1_OverrideValue: BOOL; // Frånluftsspjäll
    T_QM2_Override: BOOL; // Tilluftsspjäll
    T_QM2_OverrideValue: BOOL; // Tilluftsspjäll
    R_QM1_Override: BOOL; // Återluftsspjäll
    R_QM1_OverrideValue: BOOL; // Återluftsspjäll
    F_QM2_Override: BOOL; // Brandspjäll förbigång
    F_QM2_OverrideValue: BOOL; // Brandspjäll förbigång
    T_QM1_1_Override: BOOL; // Sektionsavfrostning
    T_QM1_1_OverrideValue: BOOL; // Sektionsavfrostning
    T_QM1_2_Override: BOOL; // Sektionsavfrostning
    T_QM1_2_OverrideValue: BOOL; // Sektionsavfrostning
    T_QM1_3_Override: BOOL; // Sektionsavfrostning
    T_QM1_3_OverrideValue: BOOL; // Sektionsavfrostning
    T_QM1_4_Override: BOOL; // Sektionsavfrostning
    T_QM1_4_OverrideValue: BOOL; // Sektionsavfrostning
    T_QM1_5_Override: BOOL; // Sektionsavfrostning
    T_QM1_5_OverrideValue: BOOL; // Sektionsavfrostning
    T_QM1_6_Override: BOOL; // Sektionsavfrostning
    T_QM1_6_OverrideValue: BOOL; // Sektionsavfrostning
    T_RUN_Override: BOOL; // Supply running (Aktiveras om tilluftsfläkten går)
    T_RUN_OverrideValue: BOOL; // Supply running (Aktiveras om tilluftsfläkten går)
    F_RUN_Override: BOOL; // Exhaust running (Aktiveras om frånluftsfläkten går)
    F_RUN_OverrideValue: BOOL; // Exhaust running (Aktiveras om frånluftsfläkten går)
	P2_Override: BOOL;
	P2_OverrideValue: BOOL;
	
	AL_A_Override: BOOL; // A-larm
	AL_A_OverrideValue: BOOL; // A-larm
	AL_B_Override: BOOL; // B-larm
	AL_B_OverrideValue: BOOL; // B-larm
	AL_C_Override: BOOL; // C-larm
	AL_C_OverrideValue: BOOL; // C-larm
	AL_D_Override: BOOL; // D-larm
	AL_D_OverrideValue: BOOL; // D-larm
END_STRUCT
END_TYPE

// ---- DUTs/Parameters/IO/DigitalOutputParameters.TcDUT
TYPE DigitalOutputParameters :
STRUCT
    H_GP1: BOOL; // Cirkulationspump värmekrets
    C_GP1: BOOL; // Cirkulationspump kylkrets
    T_QM2: BOOL; // Tilluftsspjäll
    R_QM1: BOOL; // Återluftsspjäll
    T_QM1_1: BOOL; // Sektionsavfrostning
    T_QM1_2: BOOL; // Sektionsavfrostning
    T_QM1_3: BOOL; // Sektionsavfrostning
    T_QM1_4: BOOL; // Sektionsavfrostning
    T_QM1_5: BOOL; // Sektionsavfrostning
    T_QM1_6: BOOL; // Sektionsavfrostning
    F_QM1: BOOL; // Frånluftsspjäll
    F_QM2: BOOL; // Brandspjäll förbigång
	F_QM2_ActiveWhenStopped: BOOL;
    T_RUN: BOOL; // Supply running (Aktiveras om tilluftsfläkten går)
    F_RUN: BOOL; // Exhaust running (Aktiveras om frånluftsfläkten går)
	
	AL_A: BOOL; // A-larm
	AL_B: BOOL; // B-larm
	AL_C: BOOL; // C-larm
	AL_D: BOOL; // D-larm
END_STRUCT
END_TYPE

// ---- DUTs/Parameters/IO/InputStatus.TcDUT
TYPE InputStatus :
STRUCT
    AI01: STRING;
    AI02: STRING;
    AI03: STRING;
    AI04: STRING;
    AI05: STRING;
    AI06: STRING;
    AI07: STRING;
    AI08: STRING;
    AI09: STRING;
    AI10: STRING;
    AI11: STRING;
    AI12: STRING;
    AI13: STRING;
    AI14: STRING;
    AI15: STRING;
    AI16: STRING;
    AI17: STRING;
    AI18: STRING;
    AI19: STRING;
    AI20: STRING;
    AI21: STRING;
    AI22: STRING;
    AI23: STRING;
    AI24: STRING;
END_STRUCT
END_TYPE

// ---- DUTs/Parameters/IO/IoParameters.TcDUT
TYPE IoParameters :
STRUCT
	DIn: DigitalInputParameters;
	DInLevels: DigitalInputLevels;
	DOut: DigitalOutputParameters;
	DOutOverride: DigitalOutputOverrideParameters;
	AIn: AnalogInputParameters;
	AOut: AnalogOutputParameters;
	AOutOverride: AnalogOutputOverrideParameters;
	AOutCalibration: AnalogOutputCalibration;
	Status: IoStatus;
END_STRUCT
END_TYPE

// ---- DUTs/Parameters/IO/IoStatus.TcDUT
TYPE IoStatus :
STRUCT
	SensorStatus: SensorStatus;
	InputStatus: InputStatus;
END_STRUCT
END_TYPE

// ---- DUTs/Parameters/IO/SensorStatus.TcDUT
TYPE SensorStatus :
STRUCT
	F_BT1: STRING; 
    T_BT2: STRING;
    T_BT3: STRING;
    H_BT1: STRING;
    T_BT1: STRING; 
    BT1: STRING;
    BT2: STRING;
    F_BT2: STRING;	
    F_BP1: STRING;
    T_BP1: STRING;
    F_BP2: STRING;
    T_BP2: STRING;
    F_BP3: STRING;
    T_BF1: STRING;
    F_BF1: STRING;	
END_STRUCT
END_TYPE

// ---- DUTs/Parameters/IO/SmokeControlStatus.TcDUT
TYPE SmokeControlStatus :
STRUCT
	Gateway: STRING;
	Device1: STRING;
	Device2: STRING;
	Device3: STRING;
	Device4: STRING;
END_STRUCT
END_TYPE

// ---- DUTs/Parameters/Redundancy/RedundancyParameters.TcDUT
TYPE RedundancyParameters :
STRUCT
END_STRUCT
END_TYPE

// ---- DUTs/Parameters/Regulation/AirParameters.TcDUT
TYPE AirParameters :
STRUCT
	ControlMode: FanControlTypes;
	Control: ControllerParameters;
	Defaults: DefaultParameters;
	KFactor: LREAL := 96.7;
	SlaveOffset: LREAL;
	Test1: LREAL;
	Test2: LREAL;
	Test3: LREAL;
	Test4: LREAL;
	Test5: LREAL;
	Test6: LREAL := 12345;
	ConstOutput: LREAL; // $(unit %)
	MinSpeed: LREAL := 0.0; // $(scale "0 1 0 100", unit "%", step 0.5, min 0, max 100)
	MaxSpeed: LREAL := 1.0; // $(scale "0 1 0 100", unit "%", step 0.5, min 0, max 100)
	StartupFanSpeed: LREAL;
	SetPointAdjustment: SetPointAdjustment;
	FireExhaust: FireParameters;
	FireSupply: FireParameters;
	FanType: FanTypes := FanTypes.EBM;
	SpecificFanPower: LREAL; // $(unit "kPa")
	Flow: LREAL; // $(unit "l/s")
	Power: LREAL; // $(unit "W")
	Speed: LREAL; // $(unit "rpm")
	FanEfficiency: LREAL; // $(scale "0 1 0 100", unit "%")
	PressureRise: LREAL; // $(unit "Pa")
	AdjustCSP: LREAL := 1.0; // $(skip) Adjust CSP during defrost
END_STRUCT
END_TYPE

// ---- DUTs/Parameters/Regulation/ColdRecyclingParameters.TcDUT
TYPE ColdRecyclingParameters :
STRUCT
	EN: BOOL := FALSE;
	Offset: LREAL := -2; // Cold recylcing offset (normally negative)
	Hysteresis: lreal := 0.5;
END_STRUCT
END_TYPE

// ---- DUTs/Parameters/Regulation/ControllerParameters.TcDUT
TYPE ControllerParameters :
STRUCT
	PV: LREAL;
	SP: LREAL; // $(write 0, setup, read 0, decimals 1, step 0.5)
	SP_HighSpeed: LREAL;
	CSP: LREAL;	// Beräknat börvärde
	P: LREAL := 2; // $(write 1, setup, read 0, decimals 3, step 0.001)
	I: TIME := T#2M; // $(write 1, setup, read 0, time "m:s")
	D: TIME := T#10m; // $(write 1, setup, read 0, time "m:s")
	CV: LREAL;
END_STRUCT
END_TYPE

// ---- DUTs/Parameters/Regulation/DefaultParameters.TcDUT
TYPE DefaultParameters :
STRUCT
	Pressure: ControllerParameters := ( P := 2, I := T#2M );
	Flow: ControllerParameters := ( P := 0.2, I := T#20S );
	SlaveFlow: ControllerParameters := ( P := 0.2, I := T#20S );
	Const: ControllerParameters := ( P := 1, I := T#1M );
END_STRUCT
END_TYPE

// ---- DUTs/Parameters/Regulation/FanTypes.TcDUT
{attribute 'qualified_only'}
{attribute 'strict'}
TYPE FanTypes :
(
	EBM := 0, Gebhardt
);
END_TYPE

// ---- DUTs/Parameters/Regulation/FireParameters.TcDUT
TYPE FireParameters :
STRUCT
	EN: BOOL := FALSE; // Run fan when FIRE
	Speed: LREAL := 0.8; // Speed when in FIRE (0-1)
END_STRUCT
END_TYPE

// ---- DUTs/Parameters/Regulation/HeaterOutputDirections.TcDUT
{attribute 'qualified_only'}
{attribute 'strict'}
TYPE HeaterOutputDirections :
(
	IncreaseToHeat := 0, DecreaseToHeat
);
END_TYPE

// ---- DUTs/Parameters/Regulation/RegulationControlParameters.TcDUT
TYPE RegulationControlParameters :
STRUCT
	EN: BOOL := TRUE;
	ENO: BOOL;
	//StartupHeatRecoveryTime: TIME := T#2M;
	//PostFireVentilationTime: TIME;
	//PostVentilationTime: TIME := T#2M;
END_STRUCT
END_TYPE

// ---- DUTs/Parameters/Regulation/RegulationParameters.TcDUT
TYPE RegulationParameters :
STRUCT
	Control: RegulationControlParameters;
	//SupplyAir: AirParameters := (StartupFanSpeed := 0.3, SetPointAdjustment := (Curve := (Y1 := 165, Y2 := 165, Y3 := 165, Y4 := 165, Y5 := 165, Y6 := 165, Y7 := 165, Y8 := 165, Y9 := 165)));
	//ExtractAir: AirParameters := (StartupFanSpeed := 0.4, SetPointAdjustment := (Curve := (Y1 := 160, Y2 := 160, Y3 := 160, Y4 := 160, Y5 := 160, Y6 := 160, Y7 := 160, Y8 := 160, Y9 := 160)));
	SupplyAir: AirParameters := (StartupFanSpeed := 0.3);
	ExtractAir: AirParameters := (StartupFanSpeed := 0.4);
	Temperature: TemperatureControlParameters;
	NightCoolingLimit: LREAL := 14;
	NightCoolingRequest: BOOL;
	NightCooling: BOOL;
	TemperatureCompensationSource: TemperatureCompensationSources;
	CurrentTemperatureCompensationSource: TemperatureCompensationSources;
	CompensationTemperature: LREAL;
	SystemSpecificFanPower: LREAL; // $(unit "kPa")
	SystemEfficiency: LREAL; // $(scale "0 1 0 100", unit "%")
	ApplyAbsoluteSetPointCurves: word; // $(skip)
	LastApplyAbsoluteSetPointCurves: WORD; // $(skip)
	SaveDefaults: BOOL := TRUE;
END_STRUCT
END_TYPE

// ---- DUTs/Parameters/Regulation/SetPointAdjustment.TcDUT
TYPE SetPointAdjustment :
STRUCT
	X: REAL;
	Y: REAL;
	Curve: SetPointOffsetCurve;
END_STRUCT
END_TYPE

// ---- DUTs/Parameters/Regulation/SetPointOffsetCurve.TcDUT
TYPE SetPointOffsetCurve :
STRUCT
	X1: REAL := -20;
	Y1: REAL;
	X2: REAL := -15;
	Y2: REAL;
	X3: REAL := -10;
	Y3: REAL;
	X4: REAL := -5;
	Y4: REAL;
	X5: REAL := 0;
	Y5: REAL;
	X6: REAL := 5;
	Y6: REAL;
	X7: REAL := 10;
	Y7: REAL;
	X8: REAL := 15;
	Y8: REAL;
	X9: REAL := 20;
	Y9: REAL;
END_STRUCT
END_TYPE

// ---- DUTs/Parameters/Regulation/TemperatureCompensationSources.TcDUT
{attribute 'qualified_only'}
{attribute 'strict'}
TYPE TemperatureCompensationSources :
(
	Auto := 0, BT1, T_BT2
);
END_TYPE

// ---- DUTs/Parameters/Regulation/TemperatureControlParameters.TcDUT
TYPE TemperatureControlParameters :
STRUCT
	EN: BOOL := TRUE;
	TemperatureControlSource: TemperatureControlSources;
	HeaterOutputDirection: HeaterOutputDirections := HeaterOutputDirections.DecreaseToHeat;
	//SetPointAdjustment: SetPointAdjustment := ( Curve := (Y1 := 20, Y2 := 20, Y3 := 20, Y4 := 20, Y5 := 20, Y6 := 20, Y7 := 20, Y8 := 20, Y9 := 20));
	SetPointAdjustment: SetPointAdjustment;
	Control: ControllerParameters := ( SP := 20, P := 10, I := T#2M );
	FreezeProtectionControl: ControllerParameters;
	ColdRecycling: ColdRecyclingParameters;
	Efficiency: LREAL;
	FreezeGuardLimit: REAL := 15; 
	FreezeGuardHysteresis: REAL := 1; 
	FreezeGuardControl: ControllerParameters := ( SP := 15, P := 20, I := T#30s ); 
END_STRUCT
END_TYPE

// ---- DUTs/Parameters/Regulation/TemperatureControlSources.TcDUT
{attribute 'qualified_only'}
{attribute 'strict'}
TYPE TemperatureControlSources :
(
	T_BT1 := 0, F_BT1, BT2
);
END_TYPE

// ---- DUTs/Parameters/Simulation/SimulationParameters.TcDUT
TYPE SimulationParameters :
STRUCT
	EN: BOOL;
	ENO: BOOL;
	TestSim: BOOL;
	SimCounter: INT;
END_STRUCT
END_TYPE

// ---- DUTs/Parameters/SmokeControl/NetLinkParameters.TcDUT
TYPE NetLinkParameters :
STRUCT
	{attribute 'TcEncoding':='UTF-8'}
	ModbusTCP_IP: STRING := '192.168.1.235';
	EN: BOOL := FALSE;
	Exercise: SmokeControlExerciseParameters;
	Fire: SmokeControlFireParameters;
	Error: BOOL := FALSE;
END_STRUCT
END_TYPE

// ---- DUTs/Parameters/SmokeControl/SmokeControlExerciseParameters.TcDUT
TYPE SmokeControlExerciseParameters :
STRUCT
	Interval: INT := 48; (* Central exercise interval for all damper modules (set to zero for no exercising) $(unit hour) *)
	StopVentilation: BOOL := TRUE; (* Stop ventilation during central exercise *)
	Hour: INT := 10; (* Central exercise at this hour $(unit hour) *)
	Minute: INT := 30; (* Central exercise at this minute $(unit minute) *)
END_STRUCT
END_TYPE

// ---- DUTs/Parameters/SmokeControl/SmokeControlFireParameters.TcDUT
TYPE SmokeControlFireParameters :
STRUCT
	EN: BOOL := TRUE;
END_STRUCT
END_TYPE

// ---- DUTs/Parameters/SmokeControl/SmokeControlParametersBase.TcDUT
TYPE SmokeControlParametersBase :
STRUCT
	NetLink: NetLinkParametersFB;
	DamperModules: SxDuoParameters;
END_STRUCT
END_TYPE

// ---- DUTs/Parameters/SmokeControl/SxDuoCommand.TcDUT
TYPE SxDuoCommand :
STRUCT
	ActivateFireAlarm: BOOL;
	ResetSmokeDetector: BOOL;
	ForceExercise: BOOL;	
END_STRUCT
END_TYPE

// ---- DUTs/Parameters/SmokeControl/SxDuoParameters.TcDUT
TYPE SxDuoParameters :
STRUCT
	Unit01: SxDuoUnit := ( EN := TRUE, UnitID := 21 );
	Unit02: SxDuoUnit := ( EN := FALSE, UnitID := 22 );
	Unit03: SxDuoUnit := ( EN := FALSE, UnitID := 23 );
	Unit04: SxDuoUnit := ( EN := FALSE, UnitID := 24 );
	Unit05: SxDuoUnit := ( EN := FALSE, UnitID := 25 );
	Unit06: SxDuoUnit := ( EN := FALSE, UnitID := 26 );
	Unit07: SxDuoUnit := ( EN := FALSE, UnitID := 27 );
	Unit08: SxDuoUnit := ( EN := FALSE, UnitID := 28 );
	Unit09: SxDuoUnit := ( EN := FALSE, UnitID := 29 );
	Unit10: SxDuoUnit := ( EN := FALSE, UnitID := 30 );
	Unit11: SxDuoUnit := ( EN := FALSE, UnitID := 31 );
	Unit12: SxDuoUnit := ( EN := FALSE, UnitID := 32 );
	Unit13: SxDuoUnit := ( EN := FALSE, UnitID := 33 );
	Unit14: SxDuoUnit := ( EN := FALSE, UnitID := 34 );
	Unit15: SxDuoUnit := ( EN := FALSE, UnitID := 35 );
END_STRUCT
END_TYPE

// ---- DUTs/Parameters/SmokeControl/SxDuoStatus.TcDUT
TYPE SxDuoStatus :
STRUCT
	FireAlarm: BOOL;
	Damper1Alarm: BOOL;
	Exercising: BOOL;
	Damper2Alarm: BOOL;
	Damper1Open: BOOL;
	Damper1Closed: BOOL;
	Damper2Open: BOOL;
	Damper2Closed: BOOL;
	ServiceAlarm: BOOL;
END_STRUCT
END_TYPE

// ---- DUTs/Parameters/SmokeControl/SxDuoUnit.TcDUT
TYPE SxDuoUnit :
STRUCT
	EN: BOOL;
	UnitID: BYTE;
	CentralFireAlarm: BOOL;
	CloseOnCentralFireAlarm: BOOL;
	SxDuoStatus: SxDuoStatus;
	ENO: BOOL;
	Error: BOOL;
	Fire: BOOL;
	{attribute 'TcEncoding':='UTF-8'}
	Text: STRING;
	Text_CP1252: STRING;
	SxDuoCommand: SxDuoCommand;
END_STRUCT
END_TYPE

// ---- DUTs/Parameters/System/Defrost/DefrostParameters.TcDUT
TYPE DefrostParameters :
STRUCT
	EN: BOOL := FALSE; // $(setup)
	ENO: BOOL;
	
	T_QM1_1: BOOL;
	T_QM1_2: BOOL;
	T_QM1_3: BOOL;
	T_QM1_4: BOOL;
	T_QM1_5: BOOL;
	T_QM1_6: BOOL;
	
	Sections: INT := 4; // $(setup)
	DefrostTemperature: LREAL := -40; // $(setup)
	
	SectionTime: TIME := T#10M; // $(setup)
	
	CurrentStage: INT;
	CurrentSection: DefrostSections;
	CurrentPressureLimit: LREAL;

	DefrostState: DefrostStates;
	Stage1: DefrostStageParameters := (PressureLimit := 100, SupplyAir := 0.8, ExtractAir := 1);
	Stage2: DefrostStageParameters := (PressureLimit := 150, SupplyAir := 0.4, ExtractAir := 1);
	Stage3: DefrostStageParameters := (PressureLimit := 200, SupplyAir := 0, ExtractAir := 0.5);
	
	CurrentTime: LTIME;
	//SetPointReduction: SetPointReductionParameters;
	//ExtendedDefrost: ExtendedDefrostParameters;
	//WinterShutdown: WinterShutdownParameters;
	
END_STRUCT
END_TYPE

// ---- DUTs/Parameters/System/Defrost/DefrostStageParameters.TcDUT
TYPE DefrostStageParameters :
STRUCT
	EN: BOOL := TRUE; // $(setup)
	PressureLimit: LREAL := 100; // $(setup)
	SupplyAir: LREAL := 1.0; // $(setup)
	ExtractAir: LREAL := 1.0; // $(setup)
END_STRUCT
END_TYPE

// ---- DUTs/Parameters/System/Defrost/SetPointReductionParameters.TcDUT
TYPE SetPointReductionParameters :
STRUCT
	Reduction: LREAL;
	TurnOffDelay: LTIME;
END_STRUCT
END_TYPE

// ---- DUTs/Parameters/System/Defrost/WinterShutdownParameters.TcDUT
TYPE WinterShutdownParameters :
STRUCT
	EN: BOOL;
	OutdoorTemperatureLimit: LREAL;
END_STRUCT
END_TYPE

// ---- DUTs/Parameters/System/Exercise/ExerciseCirculationPumpsParameters.TcDUT
TYPE ExerciseCirculationPumpsParameters :
STRUCT
	Interval: INT := 24; (* Central exercise interval for all damper modules (set to zero for no exercising) $(unit hour) *)
	StopVentilation: BOOL := FALSE; (* Stop ventilation during central exercise *)
	Hour: INT := 10; (* Central exercise at this hour $(unit hour) *)
	Minute: INT := 30; (* Central exercise at this minute $(unit minute) *)
	(*
	TimeChannel: TimeChannelSettings;
	StartManualExercise: BOOL;
	ExerciseStatus: BOOL;
	*)
END_STRUCT
END_TYPE

// ---- DUTs/Parameters/System/Exercise/ExerciseExternalFireControlParameters.TcDUT
TYPE ExerciseExternalFireControlParameters :
STRUCT
	TimeChannel: TimeChannelSettings;
	StartManualExercise: BOOL;
	ExerciseStatus: BOOL;
	Monitor: BOOL;
END_STRUCT
END_TYPE

// ---- DUTs/Parameters/System/Exercise/ExerciseFireBypassDamperParameters.TcDUT
TYPE ExerciseFireBypassDamperParameters :
STRUCT
	Interval: INT := 336; (* Central exercise interval for all damper modules (set to zero for no exercising) $(unit hour) *)
	StopVentilation: BOOL := TRUE; (* Stop ventilation during central exercise *)
	Hour: INT := 10; (* Central exercise at this hour $(unit hour) *)
	Minute: INT := 30; (* Central exercise at this minute $(unit minute) *)
END_STRUCT
END_TYPE

// ---- DUTs/Parameters/System/Exercise/ExerciseParameters.TcDUT
TYPE ExerciseParameters :
STRUCT
	CirculationPumps: ExerciseCirculationPumpsParameters;
	FireBypassDamper: ExerciseFireBypassDamperParameters;
	//ExternalFireControl: ExerciseExternalFireControlParameters;
	//Exercising: BOOL;
END_STRUCT
END_TYPE

// ---- DUTs/Parameters/System/Operation/AlternativeOperation.TcDUT
TYPE AlternativeOperation :
STRUCT
	EN: BOOL;
	Polarity: BOOL;
	ActivateViaDI: BOOL;
	ActivateViaADS: BOOL;
	SPTemperature: LREAL;
	UseSPTemperature: BOOL;
	SPSupplyAirPressure: LREAL;
	SPExtractAirPressure: LREAL;
	SPSupplyAirFlow: LREAL;
	SPExtractAirFlow: LREAL;
	StopUnit: BOOL;
	UnitOperation: UnitOperation;
END_STRUCT
END_TYPE

// ---- DUTs/Parameters/System/Operation/CoolingRecycling.TcDUT
TYPE CoolingRecycling :
STRUCT
	EN: BOOL := TRUE;
END_STRUCT
END_TYPE

// ---- DUTs/Parameters/System/Operation/DIStartUnit.TcDUT
TYPE DIStartUnit :
STRUCT
	SetPoints: SetPointTypes;
END_STRUCT
END_TYPE

// ---- DUTs/Parameters/System/Operation/LocalTimeControl.TcDUT
TYPE LocalTimeControl :
STRUCT
	MondayStart: DT;
	MondayStop: DT;
	TuesdayStart: DT;
	TuesdayStop: DT;
	WednesdayStart: DT;
	WednesdayStop: DT;
	ThursdayStart: DT;
	ThursdayStop: DT;
	FridayStart: DT;
	FridayStop: DT;
	SaturdayStart: DT;
	SaturdayStop: DT;
	SundayStart: DT;
	SundaydayStop: DT;
END_STRUCT
END_TYPE

// ---- DUTs/Parameters/System/Operation/MaxFilterPressure.TcDUT
TYPE MaxFilterPressure :
STRUCT
	LimitPressure: LREAL;
	OpenOnFilterAlarm: BOOL;
END_STRUCT
END_TYPE

// ---- DUTs/Parameters/System/Operation/NightReduction.TcDUT
TYPE NightReduction :
STRUCT
	EN: BOOL;
	StartTime: DT;
	StopTime: DT;
	SupplyAirFan: LREAL;
	ExtractAitFan: LREAL;
END_STRUCT
END_TYPE

// ---- DUTs/Parameters/System/Operation/OvkActivation.TcDUT
TYPE OvkActivation :
STRUCT
	Status: BOOL;
	Timeout: LTIME;
END_STRUCT
END_TYPE

// ---- DUTs/Parameters/System/Operation/RecirculationControl.TcDUT
TYPE RecirculationControl :
STRUCT
	AllowOutdoorStartViaADS: BOOL;
	Inactive: BOOL;
	OutdoorTemperatureLimit: LREAL;
	OutdoorTemperatureHysteresis: LREAL;
	SupplyAirFlow: LREAL;
	StartTime: DT;
	StopTime: DT;
	UseRecirculation: BOOL;
	AllowIndoorStartViaADS: BOOL;
	IndoorTemperatureLimit: LREAL;
	IndoorTemperatureHysteresis: LREAL;
END_STRUCT
END_TYPE

// ---- DUTs/Parameters/System/Operation/RelativeHumidity.TcDUT
TYPE RelativeHumidity :
STRUCT
	UseSioxY04: BOOL;
END_STRUCT
END_TYPE

// ---- DUTs/Parameters/System/Operation/SetPointTypes.TcDUT
{attribute 'qualified_only'}
{attribute 'strict'}
TYPE SetPointTypes :
(
	Standard := 0, Alternative
);
END_TYPE

// ---- DUTs/Parameters/System/Operation/StartControl.TcDUT
TYPE StartControl :
STRUCT
	UseLocalTimeControl: BOOL;
	UseRemoteControl: BOOL;
	RemoteControlStart: BOOL;
END_STRUCT
END_TYPE

// ---- DUTs/Parameters/System/Operation/StartupFanDelay.TcDUT
TYPE StartupFanDelay :
STRUCT
	SupplyFan: LTIME;
	ExtractFan: LTIME;
END_STRUCT
END_TYPE

// ---- DUTs/Parameters/System/Operation/StartupRecycling.TcDUT
TYPE StartupRecycling :
STRUCT
	EN: BOOL;
	Duration: LTIME;
	Speed: LREAL;
END_STRUCT
END_TYPE

// ---- DUTs/Parameters/System/Operation/SystemOperationParameters.TcDUT
TYPE SystemOperationParameters :
STRUCT
	EN: BOOL := TRUE;	// Enable the GreenMaster unit |||| Aktivera GreenMaster-enheten
	ENO: BOOL; // The GreenMaster unit is running
	RemoteEN: BOOL := TRUE;
	RemoteStart : SystemStatesRunModeExternal:=SystemStatesRunModeExternal.Auto;
	Mode:SystemStatesRunMode;
	IoUpdateEN: BOOL := TRUE; // Update inputs and outputs
	Simulation: BOOL := FALSE;
	FireDamperUsed: BOOL := TRUE;
	State: SystemStates; // Operation state
	{attribute 'TcEncoding':='UTF-8'}
	SystemName: STRING := 'GM'; // System name |||| Systemnamn
	StartupHeatRecoveryTime: TIME := TIME#3M;
	ExhaustFanStartupDelay: TIME := TIME#0S;
	SupplyFanStartupDelay: TIME := TIME#1M;
	PostVentilationTime: TIME := TIME#2M;
	PostFireVentilationTime: TIME := TIME#0M;
	TimeChannels: TimeChannelParameters;
	StartupDamperWaitTime: TIME := TIME#1M;
END_STRUCT
END_TYPE

// ---- DUTs/Parameters/System/Operation/SystemOperationParametersXXL.TcDUT
TYPE SystemOperationParametersXXL :
STRUCT
	VentilationEN: BOOL := TRUE;	// Enable the ventilation
	VentilationENO: BOOL; // The ventilation is running
END_STRUCT
END_TYPE

// ---- DUTs/Parameters/System/Operation/TimeChannelDayParameters.TcDUT
TYPE TimeChannelDayParameters :
STRUCT
	Timer1: TimeChannel1CH;
	Timer2: TimeChannel1CH;
	Timer3: TimeChannel1CH;
END_STRUCT
END_TYPE

// ---- DUTs/Parameters/System/Operation/TimeChannelParameters.TcDUT
TYPE TimeChannelParameters :
STRUCT
	TC01: TimeChannel1CH_Data := ( Day := TimerDays.Monday, OffTime := 2400 );
	TC02: TimeChannel1CH_Data := ( Day := TimerDays.Tuesday, OffTime := 2400 );
	TC03: TimeChannel1CH_Data := ( Day := TimerDays.Wednesday, OffTime := 2400 );
	TC04: TimeChannel1CH_Data := ( Day := TimerDays.Thursday, OffTime := 2400 );
	TC05: TimeChannel1CH_Data := ( Day := TimerDays.Friday, OffTime := 2400 );
	TC06: TimeChannel1CH_Data := ( Day := TimerDays.Saturday, OffTime := 2400 );
	TC07: TimeChannel1CH_Data := ( Day := TimerDays.Sunday, OffTime := 2400 );
	TC11: TimeChannel1CH_Data := ( Day := TimerDays.Monday );
	TC12: TimeChannel1CH_Data := ( Day := TimerDays.Tuesday );
	TC13: TimeChannel1CH_Data := ( Day := TimerDays.Wednesday );
	TC14: TimeChannel1CH_Data := ( Day := TimerDays.Thursday );
	TC15: TimeChannel1CH_Data := ( Day := TimerDays.Friday );
	TC16: TimeChannel1CH_Data := ( Day := TimerDays.Saturday );
	TC17: TimeChannel1CH_Data := ( Day := TimerDays.Sunday );
	TC21: TimeChannel1CH_Data := ( Day := TimerDays.Monday, Speed := 2 );
	TC22: TimeChannel1CH_Data := ( Day := TimerDays.Tuesday, Speed := 2 );
	TC23: TimeChannel1CH_Data := ( Day := TimerDays.Wednesday, Speed := 2 );
	TC24: TimeChannel1CH_Data := ( Day := TimerDays.Thursday, Speed := 2 );
	TC25: TimeChannel1CH_Data := ( Day := TimerDays.Friday, Speed := 2 );
	TC26: TimeChannel1CH_Data := ( Day := TimerDays.Saturday, Speed := 2 );
	TC27: TimeChannel1CH_Data := ( Day := TimerDays.Sunday, Speed := 2 );
	Q: BOOL; // Result of the time channels
	HighSpeed: BOOL; // Speed result of the time channels
END_STRUCT
END_TYPE

// ---- DUTs/Parameters/System/Operation/UnitOperation.TcDUT
{attribute 'qualified_only'}
{attribute 'strict'}
TYPE UnitOperation :
(
	NormalOperation := 0, AlwaysStart
);
END_TYPE

// ---- DUTs/Parameters/System/SystemParameters.TcDUT
TYPE SystemParameters :
STRUCT
	Operation: SystemOperationParameters;
	Defrost: DefrostParameters;
	Exercise: ExerciseParameters;
	SystemTime: STRING;
	ProjectDefaultSet: BOOL;
	{attribute 'TcEncoding':='UTF-8'}
	Diagram: string[80];
END_STRUCT
END_TYPE

// ---- DUTs/Parameters/System/SystemParametersXXL.TcDUT
// A bit of comment
TYPE SystemParametersXXL :
STRUCT
	Operation: SystemOperationParametersXXL;
END_STRUCT
END_TYPE

// ---- DUTs/System/Permissions.TcDUT
{attribute 'qualified_only'}
{attribute 'strict'}
TYPE Permissions :
(
	User := 0, AdminUser, SuperUser
);
END_TYPE

// ---- DUTs/System/User.TcDUT
TYPE User :
STRUCT
	{attribute 'TcEncoding':='UTF-8'}
	Email: STRING;
	{attribute 'TcEncoding':='UTF-8'}
	Password: STRING(30);
	{attribute 'TcEncoding':='UTF-8'}
	Name: STRING;
	{attribute 'TcEncoding':='UTF-8'}
	Phone: STRING(20);
	Permissions: Permissions;
END_STRUCT
END_TYPE

// ---- DUTs/Utilities/DeviationMonitorMode.TcDUT
{attribute 'qualified_only'}
{attribute 'strict'}
TYPE DeviationMonitorMode :
(
	Diff := 0, Above, Below
);
END_TYPE

// ---- DUTs/Utilities/TimeChannel1CH_Data.TcDUT
TYPE TimeChannel1CH_Data :
STRUCT
	EN: BOOL := TRUE;// Enable the time channel (settings must also be enabled)
	Speed            : INT;		// 0,1=normal speed, 2=high speed
	OnTime           : UINT;	(* Hour/minute value of the switch-on time on the day *)
	OffTime          : UINT;	(* Hour/minute value of the switch-off time on the day *)
	Day: TimerDays;
	SingleShot       : BOOL;	(* Resets EN after the on/off cycle is complete $(skip) *)   

	ENO: BOOL; // Set if enabled and settings are valid $(skip)
	Q: BOOL; // Result of the time channel
	Error: BOOL; // Settings error
	ErrorID: UDINT; // // 1 = Inconsistent weekday settings, 2 = Bad time settings, 3 = on and off times equal $(skip)
END_STRUCT
END_TYPE

// ---- DUTs/Utilities/TimeChannelSettings.TcDUT
TYPE TimeChannelSettings :
STRUCT
	EN               : BOOL;	// Enables this time channel $(skip) *)
	Speed            : INT;		// 0,1=normal speed, 2=high speed
	OnHour           : UINT;	(* Hour value of the switch-on time on the day *)
	OnMinute         : UINT;	(* Minute value of the switch-on time on the day *)
	OffHour          : UINT;	(* Hour value of the switch-off time on the day *)
	OffMinute        : UINT;	(* Minute value of the switch-off time on the day *)
	AllDays          : BOOL;	(* Selects switch-on on all days $(skip) *)       
	Monday           : BOOL;	(* ----------------------------------------------- $(skip) *)    
	Tuesday          : BOOL;	(*                                                 $(skip) *)
	Wednesday        : BOOL;	(*                                                 $(skip) *)
	Thursday         : BOOL;	(* Selects switch-on on the respective day of the week $(skip) *)
	Friday           : BOOL;	(*                                                 $(skip) *)
	Saturday         : BOOL;	(*                                                 $(skip) *)
	Sunday           : BOOL;	(* ----------------------------------------------- $(skip) *)
	SingleShot       : BOOL;	(* Resets EN after the on/off cycle is complete $(skip) *)     
	Q                : BOOL;	(* Result of the time channel $(skip) *) 
END_STRUCT
END_TYPE

// ---- DUTs/Utilities/TimerDays.TcDUT
{attribute 'qualified_only'}
{attribute 'strict'}
TYPE TimerDays :
(
	Monday := 0, Tuesday, Wednesday, Thursday, Friday, Saturday, Sunday, AllDays
);
END_TYPE

// ---- GVLs/AnalogInputs.TcDUT
TYPE AnalogInputs :
STRUCT
	// F.BT1 Frånluftstemperatur 
	AI01 AT %I*: INT;
    AI01_Error AT %I*: BOOL;
    // T.BT2 Uteluftstemperatur
	AI02 AT %I*: INT;
    AI02_Error AT %I*: BOOL;
    // T.BT3 Tilluftstemperatur (innan efterbehandling)
	AI03 AT %I*: INT;
    AI03_Error AT %I*: BOOL;
    // H.BT1 Frysskyddstemperatur (används bara om värmebatteri (av vätsketyp) är installerat)
	AI04 AT %I*: INT;
    AI04_Error AT %I*: BOOL;
    // T.BT1 Tilluftstemperatur (efter efterbehandling) 
	AI05 AT %I*: INT;
    AI05_Error AT %I*: BOOL;
    // BT1 Utomhustemperatur (extern utegivare, T.BT2 används som utegivare som standard)
	AI06 AT %I*: INT;
    AI06_Error AT %I*: BOOL;
    // BT2 Rumstemperatur (lokalgivare, används inte i bostadsaggregat)
	AI07 AT %I*: INT;
    AI07_Error AT %I*: BOOL;
    // F.BT2 Avluftstemperatur (tillval)
	AI08 AT %I*: INT;
    AI08_Error AT %I*: BOOL;
    // Reservingång (alt. T.BF1 via 0-10V) 
	AI09 AT %I*: INT;
    AI09_Error AT %I*: BOOL;
    // Reservingång (alt. F.BF1 via 0-10V)
	AI10 AT %I*: INT;
    AI10_Error AT %I*: BOOL;
    // Reservingång (alt. T.BP2 via 0-10V) 
	AI11 AT %I*: INT;
    AI11_Error AT %I*: BOOL;
    // Reservingång (alt. F.BP2 via 0-10V) 
	AI12 AT %I*: INT;
    AI12_Error AT %I*: BOOL;
    // Reservingång (alt. F.BP3 via 0-10V) 
	AI13 AT %I*: INT;
    AI13_Error AT %I*: BOOL;
    // Reservingång (alt. T.BP1 via 0-10V) 
	AI14 AT %I*: INT;
    AI14_Error AT %I*: BOOL;
    // Reservingång (alt. F.BP1 via 0-10V) 
	AI15 AT %I*: INT;
    AI15_Error AT %I*: BOOL;
    // Reservingång (extra 0-10V-ingång) 
	AI16 AT %I*: INT;
    AI16_Error AT %I*: BOOL;
	AI17 AT %I*: INT;
    AI17_Error AT %I*: BOOL;
	AI18 AT %I*: INT;
    AI18_Error AT %I*: BOOL;
	AI19 AT %I*: INT;
    AI19_Error AT %I*: BOOL;
	AI20 AT %I*: INT;
    AI20_Error AT %I*: BOOL;
	AI21 AT %I*: INT;
    AI21_Error AT %I*: BOOL;
	AI22 AT %I*: INT;
    AI22_Error AT %I*: BOOL;
	AI23 AT %I*: INT;
    AI23_Error AT %I*: BOOL;
	AI24 AT %I*: INT;
    AI24_Error AT %I*: BOOL;
END_STRUCT
END_TYPE

// ---- GVLs/AnalogOutputs.TcDUT
TYPE AnalogOutputs :
STRUCT
	// ÅV.QN1 VVX-reglering (0-10 V spjäll) 
    AO01 AT %Q*: WORD;
	//  T.GQ1 Tilluftsfläkt 
    AO02 AT %Q*: WORD;
	// F.GQ1 Frånluftsfläkt 
    AO03 AT %Q*: WORD;
	// C.QN1 Kylkrets ventil 
    AO04 AT %Q*: WORD;
	// H.QN1 Värmekrets ventil 
    AO05 AT %Q*: WORD;
	// Reservutgång
    AO06 AT %Q*: WORD;
	// Reservutgång
    AO07 AT %Q*: WORD;
	// Reservutgång
    AO08 AT %Q*: WORD;
END_STRUCT
END_TYPE

// ---- GVLs/DigitalInputs.TcDUT
TYPE DigitalInputs :
STRUCT
	// Digital Inputs, AH = active high, AL= active low
	DI01 AT %I*: BOOL; // AUTO AH (Sluten=1=Aggregat tillåts till drift via överstyrning)
	DI02 AT %I*: BOOL; // Brandlarm AL (centralt/rökdetektor frånluft)
	DI03 AT %I*: BOOL; // Utlöst AH automatsäkring, larm
	DI04 AT %I*: BOOL; // HAND AH (Sluten=Aggregat i konstant drift)
	DI05 AT %I*: BOOL; // AL Larm T.GQ1 Tilluftsfläkt
	DI06 AT %I*: BOOL; // AL Larm F.GQ1 Frånluftsfläkt
	DI07 AT %I*: BOOL; // AH F.QM2 brandspjäll ändläge 1 (spjäll stängt/normalläge)
	DI08 AT %I*: BOOL; // AL F.QM2 brandspjäll ändläge 2 (spjäll öppet/brandläge)
	DI09 AT %I*: BOOL; // Förlängd drift
	DI10 AT %I*: BOOL; // Servicelarm (centralt/rökdetektor frånluft)
	DI11 AT %I*: BOOL; // Brandlarm (tilluft)
	DI12 AT %I*: BOOL; // Servicelarm (tilluft)
	DI13 AT %I*: BOOL; // Ingång för pumpdrift, alt. pumplarm H.GP1 (värme)
	DI14 AT %I*: BOOL; // Ingång för pumpdrift, alt. pumplarm C.GP1 (kyla)
	DI15 AT %I*: BOOL; // Ingång för rotationsvakt värmeväxlare (TX1)
	DI16 AT %I*: BOOL; // Larmåterställning
	DI17 AT %I*: BOOL;
	DI18 AT %I*: BOOL;
	DI19 AT %I*: BOOL;
	DI20 AT %I*: BOOL;
	DI21 AT %I*: BOOL;
	DI22 AT %I*: BOOL;
	DI23 AT %I*: BOOL;
	DI24 AT %I*: BOOL;
	DI25 AT %I*: BOOL;
	DI26 AT %I*: BOOL;
	DI27 AT %I*: BOOL;
	DI28 AT %I*: BOOL;
	DI29 AT %I*: BOOL;
	DI30 AT %I*: BOOL;
	DI31 AT %I*: BOOL;
	DI32 AT %I*: BOOL;
END_STRUCT
END_TYPE

// ---- GVLs/DigitalInputLevels.TcDUT
TYPE DigitalInputLevels :
STRUCT
	// Digital Input Levels, false = active high
	DI01: BOOL; // AUTO AH (Sluten=1=Aggregat tillåts till drift via överstyrning)
	DI02: BOOL := TRUE; // Brandlarm AL (centralt/rökdetektor frånluft)
	DI03: BOOL := TRUE; // Utlöst AH automatsäkring, larm
	DI04: BOOL; // HAND AH (Sluten=Aggregat i konstant drift)
	DI05: BOOL := TRUE; // AL Larm T.GQ1 Tilluftsfläkt
	DI06: BOOL := TRUE; // AL Larm F.GQ1 Frånluftsfläkt
	DI07: BOOL; // AH F.QM2 brandspjäll ändläge 1 (spjäll stängt/normalläge)
	DI08: BOOL; // AL F.QM2 brandspjäll ändläge 2 (spjäll öppet/brandläge)
	DI09: BOOL; // Förlängd drift
	DI10: BOOL := TRUE; // Servicelarm (centralt/rökdetektor frånluft)
	DI11: BOOL := TRUE; // Brandlarm (tilluft)
	DI12: BOOL := FALSE; // Servicelarm (tilluft)
	DI13: BOOL; // Ingång för pumpdrift, alt. pumplarm H.GP1 (värme)
	DI14: BOOL; // Ingång för pumpdrift, alt. pumplarm C.GP1 (kyla)
	DI15: BOOL; // Ingång för rotationsvakt värmeväxlare (TX1)
	DI16: BOOL; // Larmåterställning
	DI17: BOOL;
	DI18: BOOL;
	DI19: BOOL;
	DI20: BOOL;
	DI21: BOOL;
	DI22: BOOL;
	DI23: BOOL;
	DI24: BOOL;
	DI25: BOOL;
	DI26: BOOL;
	DI27: BOOL;
	DI28: BOOL;
	DI29: BOOL;
	DI30: BOOL;
	DI31: BOOL;
	DI32: BOOL;
END_STRUCT
END_TYPE

// ---- GVLs/DigitalOutputs.TcDUT
TYPE DigitalOutputs :
STRUCT
	// H.GP1 Cirkulationspump värmekrets 
	DO01 AT %Q*: BOOL;
    //  C.GP1 Cirkulationspump kylkrets 
	DO02 AT %Q*: BOOL;
    // Exhaust running (Aktiveras om frånluftsfläkten går) 
	DO03 AT %Q*: BOOL;
    // F.QM1 Frånluftsspjäll 
	DO04 AT %Q*: BOOL;
    // T.QM3 Tilluftsspjäll 
	DO05 AT %Q*: BOOL;
    // R.QM1 Återluftsspjäll 
	DO06 AT %Q*: BOOL;
    // F.QM2 Brandspjäll förbigång 
	DO07 AT %Q*: BOOL;
    // Supply running (Aktiveras om tilluftsfläkten går) 
	DO08 AT %Q*: BOOL;
    // Sektionsavfrostningsspjäll T.QM1:1 
	DO09 AT %Q*: BOOL;
    // Sektionsavfrostningsspjäll T.QM1:2 
	DO10 AT %Q*: BOOL;
    // Sektionsavfrostningsspjäll T.QM1:3 
	DO11 AT %Q*: BOOL;
    // Sektionsavfrostningsspjäll T.QM1:4 
	DO12 AT %Q*: BOOL;
    // Sektionsavfrostningsspjäll T.QM1:5 
	DO13 AT %Q*: BOOL;
    // Sektionsavfrostningsspjäll T.QM1:6 
	DO14 AT %Q*: BOOL;
    // Reservutgång 
	DO15 AT %Q*: BOOL;
    // P2
	DO16 AT %Q*: BOOL;
	
	// A-larm
	RDO01 AT %Q*: BOOL;
    // B-larm
	RDO02 AT %Q*: BOOL;
    // C-larm
	RDO03 AT %Q*: BOOL;
    // D-larm
	RDO04 AT %Q*: BOOL;
END_STRUCT
END_TYPE

// ---- GVLs/ComponentNames.TcDUT
{attribute 'qualified_only'}
{attribute 'strict'}
{attribute 'to_string'}
TYPE ComponentNames :
(
	NONE := 0, GM, GM_BASE, GM_IO, GM_VENT, GM_XXL, GM_A, GM_C_F, GM_C_T, GM_SMOKE_CONTROL, GM_OPT_STD, SIMULATION, REDUNDANCY, EXTRA_ALARMS, SMOKE_CONTROL_ADS, PARALLEL_UNITS   
);
END_TYPE

// ---- GVLs/IOTypes.TcDUT
TYPE IOTypes :
STRUCT
	DIn: DigitalInputs;
	DOut: DigitalOutputs;
	AIn: AnalogInputs;
	AOut: AnalogOutputs;
	ModbusRTU: ModbusRTU_IO; 
END_STRUCT
END_TYPE

// ---- GVLs/Component.TcDUT
TYPE Component :
STRUCT
	Name: ComponentNames;
	{attribute 'TcEncoding':='UTF-8'}
	Path: STRING;
	Prefix: STRING;
	EN: BOOL;
	Required: BOOL;
	{attribute 'TcEncoding':='UTF-8'}
	Resource: STRING(20) := 'Parameter';
	{attribute 'TcEncoding':='UTF-8'}
	Parameters: ARRAY [0..9] OF STRING(40);
	Permissions: Permissions;
END_STRUCT
END_TYPE

// ---- GVLs/ModbusRTU_IO.TcDUT
TYPE ModbusRTU_IO :
STRUCT
	T_BP1: INT;
	T_BP1_Error: BOOL;
	F_BP1: INT;
	F_BP1_Error: BOOL;
	T_BP2: INT;
	T_BP2_Error: BOOL;
	F_BP2: INT;
	F_BP2_Error: BOOL;
	F_BP3: INT;
	F_BP3_Error: BOOL;
	T_BF1: INT;
	T_BF1_Error: BOOL;
	F_BF1: INT;	
	F_BF1_Error: BOOL;
END_STRUCT
END_TYPE

// ---- GVLs/ADS_ParallelUnits.TcGVL
{attribute 'qualified_only'}
VAR_GLOBAL
	Tags: AdsTagsParallelUnits;
END_VAR

// ---- GVLs/ADS_SmokeControl.TcGVL
{attribute 'qualified_only'}
VAR_GLOBAL PERSISTENT
	Tags: AdsTagsSmokeControl;
END_VAR

// ---- GVLs/ADS_Standard.TcGVL
{attribute 'qualified_only'}
VAR_GLOBAL PERSISTENT
	{attribute 'OPC.UA.DA' := '1'}
	Tags: AdsTags;
END_VAR

// ---- GVLs/ADS_ExtraAlarms.TcGVL
{attribute 'qualified_only'}
VAR_GLOBAL PERSISTENT
	{attribute 'OPC.UA.DA' := '1'}
	Tags: AdsTagsExtraAlarms;
END_VAR

// ---- GVLs/ExtraAlarmInputs.TcGVL
{attribute 'qualified_only'}
VAR_GLOBAL
	AL01 AT %I*: BOOL;
	AL02 AT %I*: BOOL;
	AL03 AT %I*: BOOL;
	AL04 AT %I*: BOOL;
	AL05 AT %I*: BOOL;
	AL06 AT %I*: BOOL;
	AL07 AT %I*: BOOL;
	AL08 AT %I*: BOOL;
END_VAR

// ---- GVLs/Globals.TcGVL
{attribute 'qualified_only'}
VAR_GLOBAL CONSTANT
	AlarmsLow: INT := 0;
	AlarmsHigh: INT := 99;
	EventsLow: INT := 0;
	EventsHigh: INT := 99;
END_VAR
VAR_GLOBAL
	
	// Counters
	LifeCounter: LINT;
	{attribute 'OPC.UA.DA' := '1'}
	SecondsCounter: LINT;
	SystemStartTime: DT;
	SystemUpTime: DWORD;
	{attribute 'TcEncoding':='UTF-8'}
	HostName: STRING;
	IO: IOTypes;
	AI3468: AI3468;
	ResetAlarmsCounter: INT;
END_VAR
VAR_GLOBAL PERSISTENT
	AlarmLog: AlarmLog;
	{attribute 'TcEncoding':='UTF-8'}
	AlarmLogStrings: ARRAY [AlarmsLow..AlarmsHigh] OF STRING(2000);
	EventLog: EventLogData;
	{attribute 'TcEncoding':='UTF-8'}
	EventLogStrings: ARRAY [AlarmsLow..AlarmsHigh] OF STRING(2000);
	{attribute 'TcEncoding':='UTF-8'}
	Components: STRING;
END_VAR

// ---- GVLs/GVL.TcGVL
{attribute 'qualified_only'}
VAR_GLOBAL
	mb_Input_Coils:ARRAY[0..255] OF BOOL;
	mb_Output_Coils:ARRAY[0..255] OF BOOL;
	mb_Output_Registers:ARRAY[0..2000] OF DINT;
	mb_Input_Registers:ARRAY[0..2000] OF WORD;	
END_VAR

// ---- GVLs/GVL_Redundancy.TcGVL
{attribute 'qualified_only'}
VAR_GLOBAL
	Tags: TagsRedundancy;	
END_VAR

